IF ((P2Btn.P2M1_Tricolorlamp_Yellow AND NOT P2M1_DTSysState.bErrorStop AND NOT P2M1_WJSysState.bErrorStop AND NOT P2M1_WJSysState.bErrorStop AND
    P2Btn.P2M2_Tricolorlamp_Yellow AND NOT P2M2_DTSysState.bErrorStop AND NOT P2M2_WJSysState.bErrorStop AND NOT P2M2_WJSysState.bErrorStop AND
    P2Btn.P2M3_Tricolorlamp_Yellow AND NOT P2M3_DTSysState.bErrorStop AND NOT P2M3_WJSysState.bErrorStop AND NOT P2M3_WJSysState.bErrorStop ) OR 
	((P2M1_DTSysState.bErrorStop OR P2M1_WJSysState.bErrorStop OR P2M1_WJSysState.bErrorStop) AND
    (P2Btn.P2M2_Tricolorlamp_Yellow AND NOT P2M2_DTSysState.bErrorStop AND NOT P2M2_WJSysState.bErrorStop AND NOT P2M2_WJSysState.bErrorStop) AND
	(P2Btn.P2M3_Tricolorlamp_Yellow AND NOT P2M3_DTSysState.bErrorStop AND NOT P2M3_WJSysState.bErrorStop AND NOT P2M3_WJSysState.bErrorStop)) OR
	((P2Btn.P2M1_Tricolorlamp_Yellow AND NOT P2M1_DTSysState.bErrorStop AND NOT P2M1_WJSysState.bErrorStop AND NOT P2M1_WJSysState.bErrorStop) AND
	(P2M2_DTSysState.bErrorStop OR P2M2_WJSysState.bErrorStop OR P2M2_WJSysState.bErrorStop) AND	
	(P2Btn.P2M3_Tricolorlamp_Yellow AND NOT P2M3_DTSysState.bErrorStop AND NOT P2M3_WJSysState.bErrorStop AND NOT P2M3_WJSysState.bErrorStop)) OR
	((P2Btn.P2M1_Tricolorlamp_Yellow AND NOT P2M1_DTSysState.bErrorStop AND NOT P2M1_WJSysState.bErrorStop AND NOT P2M1_WJSysState.bErrorStop) AND
	(P2Btn.P2M2_Tricolorlamp_Yellow AND NOT P2M2_DTSysState.bErrorStop AND NOT P2M2_WJSysState.bErrorStop AND NOT P2M2_WJSysState.bErrorStop) AND
	(P2M3_DTSysState.bErrorStop OR P2M3_WJSysState.bErrorStop OR P2M3_WJSysState.bErrorStop) ) OR  Standby_TON.Q) AND
	NOT P2Btn.P2M1_Tricolorlamp_Green AND NOT P2Btn.P2M2_Tricolorlamp_Green AND NOT P2Btn.P2M3_Tricolorlamp_Green THEN
	 Status_switching2_TON.IN:=TRUE ;
	 Status_switching_TON.IN:=FALSE ;
END_IF

IF  Status_switching2_TON.Q THEN 
    P3Press.Device_Status_code:=18 ; //设备待机
END_IF	

Equipment_parameter_check_R(CLK:=Equipment_parameter_check=2  , Q=> ); //Equipment_parameter_check=1参数校验OK,Equipment_parameter_check=1参数校验NG
IF Equipment_parameter_check_R.Q THEN
   P3_Error[40]:=TRUE ;	//MES校验热压、称重、测厚参数报警，请检查参数设置s是否正确
   Equipment_parameter_check:=0 ;
END_IF

//xfp20240315 与MES交互优报表

ton2(IN:=NOT ton2.Q , PT:=T#5M , Q=> , ET=> );
IF ton2.Q THEN
   Mes1.uOther[0]:=1;
END_IF
ExcelRate_R(clk:=(Mes1.uOther[0]=1),Q=>);	//MES读取触发上升沿
MTDExcelRate_R(clk:=(MTD_Mes1.uOther[0]=2),Q=>);	//MTD完成上升沿
tonWaitMQdata(pt:=T#2S);
IF ExcelRate_R.Q THEN
	Mes1RdStep:=10;
END_IF	
CASE Mes1RdStep OF
	10:
		DTM_Mes1.uOther[0]:=1;
		Mes1RdStep:=20;
	20:	
		IF MTDExcelRate_R.Q THEN
			DTM_Mes1.uOther[0]:=0;
			Mes1RdStep:=30;
		END_IF
		IF NOT tonWaitMQdata.Q THEN
			tonWaitMQdata.IN:=TRUE;
		ELSE
			tonWaitMQdata.IN:=FALSE;
			Mes1.uOther[0]:=3;
			DTM_Mes1.uOther[0]:=0;
			Mes1RdStep:=0;	
		END_IF
	30:
		tonWaitMQdata.IN:=FALSE;
		IF system.stTime.wHour >=8 AND system.stTime.wHour <20 THEN
			Mes1.rExcelRate[0]:=1;	//班次，白班
			Mes1.rExcelRate[1]:=0;
			Mes1.rExcelRate[2]:=P3_Production.HMI_DayOkCount;	//生产良品数量
			Mes1.rExcelRate[3]:=P3_Production.HMI_DayNgCount;	//生产不良品数量
			Mes1.rExcelRate[4]:=P3_Production.HMI_DayQualified;	//良率			
			Mes1.rExcelRate[5]	:=MTD_Mes1.rExcelRate[0];
			Mes1.rExcelRate[6]	:=MTD_Mes1.rExcelRate[1];
			Mes1.rExcelRate[7]	:=MTD_Mes1.rExcelRate[2];
			Mes1.rExcelRate[8]	:=MTD_Mes1.rExcelRate[3];
			Mes1.rExcelRate[9]	:=MTD_Mes1.rExcelRate[4];
			Mes1.rExcelRate[10]	:=MTD_Mes1.rExcelRate[5];
			Mes1.rExcelRate[11]	:=MTD_Mes1.rExcelRate[6];
			Mes1.rExcelRate[12]	:=MTD_Mes1.rExcelRate[7];
			Mes1.rExcelRate[13]	:=MTD_Mes1.rExcelRate[8];
			Mes1.rExcelRate[14]	:=MTD_Mes1.rExcelRate[9];
			Mes1.rExcelRate[15]	:=MTD_Mes1.rExcelRate[10];
			Mes1.rExcelRate[16]	:=MTD_Mes1.rExcelRate[11];
			Mes1.rExcelRate[17]	:=MTD_Mes1.rExcelRate[12];
			Mes1.rExcelRate[18]	:=MTD_Mes1.rExcelRate[13];
			Mes1.rExcelRate[19]	:=MTD_Mes1.rExcelRate[14];
			Mes1.rExcelRate[20]	:=MTD_Mes1.rExcelRate[15];
			Mes1.rExcelRate[21]	:=MTD_Mes1.rExcelRate[16];
			Mes1.rExcelRate[22]	:=MTD_Mes1.rExcelRate[17];
			Mes1.rExcelRate[23]	:=MTD_Mes1.rExcelRate[18];
			Mes1.rExcelRate[24]	:=MTD_Mes1.rExcelRate[19];
			Mes1.rExcelRate[25]	:=MTD_Mes1.rExcelRate[20];
			Mes1.rExcelRate[26]	:=MTD_Mes1.rExcelRate[21];
			Mes1.rExcelRate[27]	:=MTD_Mes1.rExcelRate[22];
			Mes1.rExcelRate[28]	:=MTD_Mes1.rExcelRate[23];
			Mes1.rExcelRate[29]	:=MTD_Mes1.rExcelRate[24];
			Mes1.rExcelRate[30]	:=MTD_Mes1.rExcelRate[25];
			Mes1.rExcelRate[31]	:=MTD_Mes1.rExcelRate[26];			
			Mes1.rExcelRate[32]:=User01.P2M1_CCD.AnRec.DayNgclassification.X1_NG;	//叠台一正极X1纠偏轴不良数
			Mes1.rExcelRate[33]:=User01.P2M1_CCD.AnRec.DayNgclassification.X2_NG;	//叠台一正极X2纠偏轴不良数
			Mes1.rExcelRate[34]:=User01.P2M1_CCD.AnRec.DayNgclassification.Y_NG;	//叠台一正极Y纠偏轴不良数
			Mes1.rExcelRate[35]:=User01.P2M1_CCD.AnRec.DayNgclassification.R_NG;	//叠台一正极R角轮廓不良数
			Mes1.rExcelRate[36]:=User01.P2M1_CCD.AnRec.DayNgclassification.other_NG;	//叠台一正极其他类不良数
			Mes1.rExcelRate[37]:=User01.P2M2_CCD.AnRec.DayNgclassification.X1_NG;	//叠台二正极X1纠偏轴不良数
			Mes1.rExcelRate[38]:=User01.P2M2_CCD.AnRec.DayNgclassification.X2_NG;	//叠台二正极X2纠偏轴不良数
			Mes1.rExcelRate[39]:=User01.P2M2_CCD.AnRec.DayNgclassification.Y_NG;	//叠台二正极Y纠偏轴不良数
			Mes1.rExcelRate[40]:=User01.P2M2_CCD.AnRec.DayNgclassification.R_NG;	//叠台二正极R角轮廓不良数
			Mes1.rExcelRate[41]:=User01.P2M2_CCD.AnRec.DayNgclassification.other_NG;	//叠台二正极其他类不良数
			Mes1.rExcelRate[42]:=User01.P2M3_CCD.AnRec.DayNgclassification.X1_NG;	//叠台三正极X1纠偏轴不良数
			Mes1.rExcelRate[43]:=User01.P2M3_CCD.AnRec.DayNgclassification.X2_NG;	//叠台三正极X2纠偏轴不良数
			Mes1.rExcelRate[44]:=User01.P2M3_CCD.AnRec.DayNgclassification.Y_NG;	//叠台三正极Y纠偏轴不良数
			Mes1.rExcelRate[45]:=User01.P2M3_CCD.AnRec.DayNgclassification.R_NG;	//叠台三正极R角轮廓不良数
			Mes1.rExcelRate[46]:=User01.P2M3_CCD.AnRec.DayNgclassification.other_NG;	//叠台三正极其他类不良数
			//Mes1.rExcelRate[47]:=User01.P2M1_MachCtrl.DT_b.DT_DayHough_U;	//1#叠台OH不良，NG个数
			Mes1.rExcelRate[47]:=User01.P2M1_MachCtrl.DT_b.DT_DayHoughAn;		//1#叠台OH不良，正极NG数
			//Mes1.rExcelRate[49]:=User01.P2M2_MachCtrl.DT_b.DT_DayHough_U;	//2#叠台OH不良，NG个数
			Mes1.rExcelRate[49]:=User01.P2M2_MachCtrl.DT_b.DT_DayHoughAn;		//2#叠台OH不良，正极NG数
		//	Mes1.rExcelRate[51]:=User01.P2M3_MachCtrl.DT_b.DT_DayHough_U;	//3#叠台OH不良，NG个数
			Mes1.rExcelRate[51]:=User01.P2M3_MachCtrl.DT_b.DT_DayHoughAn;		//3#叠台OH不良，正极NG数
			Mes1.rExcelRate[53]:=P3_Production.NgPerHourDayCount[2];	//hi-potNG
			Mes1.rExcelRate[54]:=P3_Production.NgPerHourDayCount[4];	//厚度NG
			Mes1.rExcelRate[55]:=P3_Production.NgPerHourDayCount[6];	//烘烤超时NG
			Mes1.rExcelRate[56]:=P3_Production.NgPerHourDayCount[5];	//MESNG
			Mes1.rExcelRate[57]:=P3_Production.NgPerHourDayCount[1];	//扫码NG
			Mes1.rExcelRate[58]:=P3_Production.NgPerHourDayCount[3];	//其他不良	
			Mes1.rExcelRate[59]	:=MTD_Mes1.rExcelRate[27];
			Mes1.rExcelRate[60]	:=MTD_Mes1.rExcelRate[28];
			Mes1.rExcelRate[61]	:=MTD_Mes1.rExcelRate[29];
			Mes1.rExcelRate[62]	:=MTD_Mes1.rExcelRate[30];
			Mes1.rExcelRate[63]	:=MTD_Mes1.rExcelRate[31];
			Mes1.rExcelRate[64]	:=MTD_Mes1.rExcelRate[32];
			Mes1.rExcelRate[65]	:=MTD_Mes1.rExcelRate[33];
			Mes1.rExcelRate[66]	:=MTD_Mes1.rExcelRate[34];
			Mes1.rExcelRate[67]	:=MTD_Mes1.rExcelRate[35];
			Mes1.rExcelRate[68]	:=MTD_Mes1.rExcelRate[36];
			Mes1.rExcelRate[69]	:=MTD_Mes1.rExcelRate[37];
			Mes1.rExcelRate[70]	:=MTD_Mes1.rExcelRate[38];
			Mes1.rExcelRate[71]	:=MTD_Mes1.rExcelRate[39];
			Mes1.rExcelRate[72]	:=MTD_Mes1.rExcelRate[40];
			Mes1.rExcelRate[73]	:=MTD_Mes1.rExcelRate[41];
			Mes1.rExcelRate[74]	:=MTD_Mes1.rExcelRate[42];
			Mes1.rExcelRate[75]	:=MTD_Mes1.rExcelRate[43];
			Mes1.rExcelRate[76]	:=MTD_Mes1.rExcelRate[44];
			Mes1.rExcelRate[77]	:=MTD_Mes1.rExcelRate[45];
			Mes1.rExcelRate[78]	:=MTD_Mes1.rExcelRate[46];
			Mes1.rExcelRate[79]	:=MTD_Mes1.rExcelRate[47];
			Mes1.rExcelRate[80]	:=MTD_Mes1.rExcelRate[48];
			Mes1.rExcelRate[81]	:=MTD_Mes1.rExcelRate[49];
			Mes1.rExcelRate[82]	:=MTD_Mes1.rExcelRate[50];
			Mes1.rExcelRate[83]	:=MTD_Mes1.rExcelRate[51];
			Mes1.rExcelRate[84]	:=MTD_Mes1.rExcelRate[52];			
			Mes1.rExcelRate[85]:=User01.P2M1_CCD.CaRec.DayNgclassification.X1_NG;	//叠台一负极X1纠偏轴不良数
			Mes1.rExcelRate[86]:=User01.P2M1_CCD.CaRec.DayNgclassification.X2_NG;	//叠台一负极X2纠偏轴不良数
			Mes1.rExcelRate[87]:=User01.P2M1_CCD.CaRec.DayNgclassification.Y_NG;	//叠台一负极Y纠偏轴不良数
			Mes1.rExcelRate[88]:=User01.P2M1_CCD.CaRec.DayNgclassification.R_NG;	//叠台一负极R角轮廓不良数
			Mes1.rExcelRate[89]:=User01.P2M1_CCD.CaRec.DayNgclassification.other_NG;	//叠台一负极其他类不良数
			Mes1.rExcelRate[90]:=User01.P2M2_CCD.CaRec.DayNgclassification.X1_NG;	//叠台二负极X1纠偏轴不良数
			Mes1.rExcelRate[91]:=User01.P2M2_CCD.CaRec.DayNgclassification.X2_NG;	//叠台二负极X2纠偏轴不良数
			Mes1.rExcelRate[92]:=User01.P2M2_CCD.CaRec.DayNgclassification.Y_NG;	//叠台二负极Y纠偏轴不良数
			Mes1.rExcelRate[93]:=User01.P2M2_CCD.CaRec.DayNgclassification.R_NG;	//叠台二负极R角轮廓不良数
			Mes1.rExcelRate[94]:=User01.P2M2_CCD.CaRec.DayNgclassification.other_NG;	//叠台二负极其他类不良数
			Mes1.rExcelRate[95]:=User01.P2M3_CCD.CaRec.DayNgclassification.X1_NG;	//叠台三负极X1纠偏轴不良数
			Mes1.rExcelRate[96]:=User01.P2M3_CCD.CaRec.DayNgclassification.X2_NG;	//叠台三负极X2纠偏轴不良数
			Mes1.rExcelRate[97]:=User01.P2M3_CCD.CaRec.DayNgclassification.Y_NG;	//叠台三负极Y纠偏轴不良数
			Mes1.rExcelRate[98]:=User01.P2M3_CCD.CaRec.DayNgclassification.R_NG;	//叠台三负极R角轮廓不良数
			Mes1.rExcelRate[99]:=User01.P2M3_CCD.CaRec.DayNgclassification.other_NG;	//叠台三负极其他类不良数			
			Mes1.rExcelRate[100]:=User01.P2M1_MachCtrl.DT_b.DT_DayHoughCa;	//1#叠台OH不良负极NG数
			Mes1.rExcelRate[101]:=User01.P2M2_MachCtrl.DT_b.DT_DayHoughCa;	//2#叠台OH不良负极NG数
			Mes1.rExcelRate[102]:=User01.P2M3_MachCtrl.DT_b.DT_DayHoughCa;	//3#叠台OH不良负极NG数
			Mes1.rExcelRate[103]	:=MTD_Mes1.rExcelRate[53];			
			Mes1.rExcelRate[104]	:=MTD_Mes1.rExcelRate[54];	
			Mes1.rExcelRate[105]	:=MTD_Mes1.rExcelRate[55];			
			Mes1.rExcelRate[106]	:=MTD_Mes1.rExcelRate[56];	
			Mes1.rExcelRate[107]	:=MTD_Mes1.rExcelRate[57];			
			Mes1.rExcelRate[108]	:=MTD_Mes1.rExcelRate[58];	
			Mes1.rExcelRate[109]	:=(MTD_Mes1.rExcelRate[0]+MTD_Mes1.rExcelRate[15])/P2M1_Par.stDT_date.An_Quantity;		
			Mes1.rExcelRate[110]	:=(MTD_Mes1.rExcelRate[27]+MTD_Mes1.rExcelRate[41])/P2M1_Par.stDT_date.Ca_Quantity;			
			Mes1.uOther[0]:=2;	//plc数据写入完成
			Mes1RdStep:=0;
		ELSIF system.stTime.wHour >=20 OR system.stTime.wHour<8 THEN
			Mes1.rExcelRate[0]:=2;	//班次，夜班
			Mes1.rExcelRate[1]:=0;
			Mes1.rExcelRate[2]:=P3_Production.HMI_NightOkCount;	//生产良品数量
			Mes1.rExcelRate[3]:=P3_Production.HMI_NightNgCount;	//生产不良品数量
			Mes1.rExcelRate[4]:=P3_Production.HMI_NightQualified;	//良率			
			Mes1.rExcelRate[5]	:=MTD_Mes1.rExcelRate[0];
			Mes1.rExcelRate[6]	:=MTD_Mes1.rExcelRate[1];
			Mes1.rExcelRate[7]	:=MTD_Mes1.rExcelRate[2];
			Mes1.rExcelRate[8]	:=MTD_Mes1.rExcelRate[3];
			Mes1.rExcelRate[9]	:=MTD_Mes1.rExcelRate[4];
			Mes1.rExcelRate[10]	:=MTD_Mes1.rExcelRate[5];
			Mes1.rExcelRate[11]	:=MTD_Mes1.rExcelRate[6];
			Mes1.rExcelRate[12]	:=MTD_Mes1.rExcelRate[7];
			Mes1.rExcelRate[13]	:=MTD_Mes1.rExcelRate[8];
			Mes1.rExcelRate[14]	:=MTD_Mes1.rExcelRate[9];
			Mes1.rExcelRate[15]	:=MTD_Mes1.rExcelRate[10];
			Mes1.rExcelRate[16]	:=MTD_Mes1.rExcelRate[11];
			Mes1.rExcelRate[17]	:=MTD_Mes1.rExcelRate[12];
			Mes1.rExcelRate[18]	:=MTD_Mes1.rExcelRate[13];
			Mes1.rExcelRate[19]	:=MTD_Mes1.rExcelRate[14];
			Mes1.rExcelRate[20]	:=MTD_Mes1.rExcelRate[15];
			Mes1.rExcelRate[21]	:=MTD_Mes1.rExcelRate[16];
			Mes1.rExcelRate[22]	:=MTD_Mes1.rExcelRate[17];
			Mes1.rExcelRate[23]	:=MTD_Mes1.rExcelRate[18];
			Mes1.rExcelRate[24]	:=MTD_Mes1.rExcelRate[19];
			Mes1.rExcelRate[25]	:=MTD_Mes1.rExcelRate[20];
			Mes1.rExcelRate[26]	:=MTD_Mes1.rExcelRate[21];
			Mes1.rExcelRate[27]	:=MTD_Mes1.rExcelRate[22];
			Mes1.rExcelRate[28]	:=MTD_Mes1.rExcelRate[23];
			Mes1.rExcelRate[29]	:=MTD_Mes1.rExcelRate[24];
			Mes1.rExcelRate[30]	:=MTD_Mes1.rExcelRate[25];
			Mes1.rExcelRate[31]	:=MTD_Mes1.rExcelRate[26];			
			Mes1.rExcelRate[32]:=User01.P2M1_CCD.AnRec.NightNgclassification.X1_NG;	//叠台一正极X1纠偏轴不良数
			Mes1.rExcelRate[33]:=User01.P2M1_CCD.AnRec.NightNgclassification.X2_NG;	//叠台一正极X2纠偏轴不良数
			Mes1.rExcelRate[34]:=User01.P2M1_CCD.AnRec.NightNgclassification.Y_NG;	//叠台一正极Y纠偏轴不良数
			Mes1.rExcelRate[35]:=User01.P2M1_CCD.AnRec.NightNgclassification.R_NG;	//叠台一正极R角轮廓不良数
			Mes1.rExcelRate[36]:=User01.P2M1_CCD.AnRec.NightNgclassification.other_NG;	//叠台一正极其他类不良数
			Mes1.rExcelRate[37]:=User01.P2M2_CCD.AnRec.NightNgclassification.X1_NG;	//叠台二正极X1纠偏轴不良数
			Mes1.rExcelRate[38]:=User01.P2M2_CCD.AnRec.NightNgclassification.X2_NG;	//叠台二正极X2纠偏轴不良数
			Mes1.rExcelRate[39]:=User01.P2M2_CCD.AnRec.NightNgclassification.Y_NG;	//叠台二正极Y纠偏轴不良数
			Mes1.rExcelRate[40]:=User01.P2M2_CCD.AnRec.NightNgclassification.R_NG;	//叠台二正极R角轮廓不良数
			Mes1.rExcelRate[41]:=User01.P2M2_CCD.AnRec.NightNgclassification.other_NG;	//叠台二正极其他类不良数
			Mes1.rExcelRate[42]:=User01.P2M3_CCD.AnRec.NightNgclassification.X1_NG;	//叠台三正极X1纠偏轴不良数
			Mes1.rExcelRate[43]:=User01.P2M3_CCD.AnRec.NightNgclassification.X2_NG;	//叠台三正极X2纠偏轴不良数
			Mes1.rExcelRate[44]:=User01.P2M3_CCD.AnRec.NightNgclassification.Y_NG;	//叠台三正极Y纠偏轴不良数
			Mes1.rExcelRate[45]:=User01.P2M3_CCD.AnRec.NightNgclassification.R_NG;	//叠台三正极R角轮廓不良数
			Mes1.rExcelRate[46]:=User01.P2M3_CCD.AnRec.NightNgclassification.other_NG;	//叠台三正极其他类不良数
		//	Mes1.rExcelRate[47]:=User01.P2M1_MachCtrl.DT_b.DT_NightHough_U;	//1#叠台OH不良，NG个数
			Mes1.rExcelRate[47]:=User01.P2M1_MachCtrl.DT_b.DT_NightHoughAn;		//1#叠台OH不良，正极NG数
		//	Mes1.rExcelRate[49]:=User01.P2M2_MachCtrl.DT_b.DT_NightHough_U;	//2#叠台OH不良，NG个数
			Mes1.rExcelRate[49]:=User01.P2M2_MachCtrl.DT_b.DT_NightHoughAn;		//2#叠台OH不良，正极NG数
		//	Mes1.rExcelRate[51]:=User01.P2M3_MachCtrl.DT_b.DT_NightHough_U;	//3#叠台OH不良，NG个数
			Mes1.rExcelRate[51]:=User01.P2M3_MachCtrl.DT_b.DT_NightHoughAn;		//3#叠台OH不良，正极NG数
			Mes1.rExcelRate[53]:=P3_Production.NgPerHourNightCount[2];	//hi-potNG
			Mes1.rExcelRate[54]:=P3_Production.NgPerHourNightCount[4];	//厚度NG
			Mes1.rExcelRate[55]:=P3_Production.NgPerHourNightCount[6];	//烘烤超时NG
			Mes1.rExcelRate[56]:=P3_Production.NgPerHourNightCount[5];	//MESNG
			Mes1.rExcelRate[57]:=P3_Production.NgPerHourNightCount[1];	//扫码NG
			Mes1.rExcelRate[58]:=P3_Production.NgPerHourNightCount[3];	//其他不良	
			Mes1.rExcelRate[59]	:=MTD_Mes1.rExcelRate[27];
			Mes1.rExcelRate[60]	:=MTD_Mes1.rExcelRate[28];
			Mes1.rExcelRate[61]	:=MTD_Mes1.rExcelRate[29];
			Mes1.rExcelRate[62]	:=MTD_Mes1.rExcelRate[30];
			Mes1.rExcelRate[63]	:=MTD_Mes1.rExcelRate[31];
			Mes1.rExcelRate[64]	:=MTD_Mes1.rExcelRate[32];
			Mes1.rExcelRate[65]	:=MTD_Mes1.rExcelRate[33];
			Mes1.rExcelRate[66]	:=MTD_Mes1.rExcelRate[34];
			Mes1.rExcelRate[67]	:=MTD_Mes1.rExcelRate[35];
			Mes1.rExcelRate[68]	:=MTD_Mes1.rExcelRate[36];
			Mes1.rExcelRate[69]	:=MTD_Mes1.rExcelRate[37];
			Mes1.rExcelRate[70]	:=MTD_Mes1.rExcelRate[38];
			Mes1.rExcelRate[71]	:=MTD_Mes1.rExcelRate[39];
			Mes1.rExcelRate[72]	:=MTD_Mes1.rExcelRate[40];
			Mes1.rExcelRate[73]	:=MTD_Mes1.rExcelRate[41];
			Mes1.rExcelRate[74]	:=MTD_Mes1.rExcelRate[42];
			Mes1.rExcelRate[75]	:=MTD_Mes1.rExcelRate[43];
			Mes1.rExcelRate[76]	:=MTD_Mes1.rExcelRate[44];
			Mes1.rExcelRate[77]	:=MTD_Mes1.rExcelRate[45];
			Mes1.rExcelRate[78]	:=MTD_Mes1.rExcelRate[46];
			Mes1.rExcelRate[79]	:=MTD_Mes1.rExcelRate[47];
			Mes1.rExcelRate[80]	:=MTD_Mes1.rExcelRate[48];
			Mes1.rExcelRate[81]	:=MTD_Mes1.rExcelRate[49];
			Mes1.rExcelRate[82]	:=MTD_Mes1.rExcelRate[50];
			Mes1.rExcelRate[83]	:=MTD_Mes1.rExcelRate[51];
			Mes1.rExcelRate[84]	:=MTD_Mes1.rExcelRate[52];			
			Mes1.rExcelRate[85]:=User01.P2M1_CCD.CaRec.NightNgclassification.X1_NG;	//叠台一负极X1纠偏轴不良数
			Mes1.rExcelRate[86]:=User01.P2M1_CCD.CaRec.NightNgclassification.X2_NG;	//叠台一负极X2纠偏轴不良数
			Mes1.rExcelRate[87]:=User01.P2M1_CCD.CaRec.NightNgclassification.Y_NG;	//叠台一负极Y纠偏轴不良数
			Mes1.rExcelRate[88]:=User01.P2M1_CCD.CaRec.NightNgclassification.R_NG;	//叠台一负极R角轮廓不良数
			Mes1.rExcelRate[89]:=User01.P2M1_CCD.CaRec.NightNgclassification.other_NG;	//叠台一负极其他类不良数
			Mes1.rExcelRate[90]:=User01.P2M2_CCD.CaRec.NightNgclassification.X1_NG;	//叠台二负极X1纠偏轴不良数
			Mes1.rExcelRate[91]:=User01.P2M2_CCD.CaRec.NightNgclassification.X2_NG;	//叠台二负极X2纠偏轴不良数
			Mes1.rExcelRate[92]:=User01.P2M2_CCD.CaRec.NightNgclassification.Y_NG;	//叠台二负极Y纠偏轴不良数
			Mes1.rExcelRate[93]:=User01.P2M2_CCD.CaRec.NightNgclassification.R_NG;	//叠台二负极R角轮廓不良数
			Mes1.rExcelRate[94]:=User01.P2M2_CCD.CaRec.NightNgclassification.other_NG;	//叠台二负极其他类不良数
			Mes1.rExcelRate[95]:=User01.P2M3_CCD.CaRec.NightNgclassification.X1_NG;	//叠台三负极X1纠偏轴不良数
			Mes1.rExcelRate[96]:=User01.P2M3_CCD.CaRec.NightNgclassification.X2_NG;	//叠台三负极X2纠偏轴不良数
			Mes1.rExcelRate[97]:=User01.P2M3_CCD.CaRec.NightNgclassification.Y_NG;	//叠台三负极Y纠偏轴不良数
			Mes1.rExcelRate[98]:=User01.P2M3_CCD.CaRec.NightNgclassification.R_NG;	//叠台三负极R角轮廓不良数
			Mes1.rExcelRate[99]:=User01.P2M3_CCD.CaRec.NightNgclassification.other_NG;	//叠台三负极其他类不良数			
			Mes1.rExcelRate[100]:=User01.P2M1_MachCtrl.DT_b.DT_NightHoughCa;	//1#叠台OH不良负极NG数
			Mes1.rExcelRate[101]:=User01.P2M2_MachCtrl.DT_b.DT_NightHoughCa;	//2#叠台OH不良负极NG数
			Mes1.rExcelRate[102]:=User01.P2M3_MachCtrl.DT_b.DT_NightHoughCa;	//3#叠台OH不良负极NG数
			Mes1.rExcelRate[103]	:=MTD_Mes1.rExcelRate[53];			
			Mes1.rExcelRate[104]	:=MTD_Mes1.rExcelRate[54];	
			Mes1.rExcelRate[105]	:=MTD_Mes1.rExcelRate[55];			
			Mes1.rExcelRate[106]	:=MTD_Mes1.rExcelRate[56];	
			Mes1.rExcelRate[107]	:=MTD_Mes1.rExcelRate[57];			
			Mes1.rExcelRate[108]	:=MTD_Mes1.rExcelRate[58];		
     		Mes1.rExcelRate[109]	:=(MTD_Mes1.rExcelRate[0]+MTD_Mes1.rExcelRate[15])/P2M1_Par.stDT_date.An_Quantity;		
			Mes1.rExcelRate[110]	:=(MTD_Mes1.rExcelRate[27]+MTD_Mes1.rExcelRate[41])/P2M1_Par.stDT_date.Ca_Quantity;	;		
			Mes1.uOther[0]:=2;	//plc数据写入完成
			Mes1RdStep:=0;
		END_IF	
END_CASE


//功能开关状态
Mes1.bFuncEN[1]:=MTD_Mes1.bFuncEN[1];//模切段CCD通讯开关状态
Mes1.bFuncEN[2]:=MTD_Mes1.bFuncEN[2];//线扫CCD开关状态
Mes1.bFuncEN[3]:=MTD_Mes1.bFuncEN[3];//冲R角定位开关状态
Mes1.bFuncEN[4]:=MTD_Mes1.bFuncEN[4];//裁切定位开关状态
Mes1.bFuncEN[5]:=MTD_Mes1.bFuncEN[5];//尺寸检测开关状态
Mes1.bFuncEN[6]:=MTD_Mes1.bFuncEN[6];//物料校验功能开关状态
Mes1.bFuncEN[7]:=MTD_Mes1.bFuncEN[7];//来料不良检测开关状态
Mes1.bFuncEN[8]:=P2M1_Par.iModeEN.CCD_ChosesHMIEN;//一叠台CCD通讯开关状态
Mes1.bFuncEN[9]:=P2M2_Par.iModeEN.CCD_ChosesHMIEN;
Mes1.bFuncEN[10]:=P2M3_Par.iModeEN.CCD_ChosesHMIEN;
Mes1.bFuncEN[11]:=P2M1_Par.iModeEN.DT_CCD_TwoModelEN;//一叠台CCD复检开关状态
Mes1.bFuncEN[12]:=P2M2_Par.iModeEN.DT_CCD_TwoModelEN;
Mes1.bFuncEN[13]:=P2M3_Par.iModeEN.DT_CCD_TwoModelEN;
Mes1.bFuncEN[14]:=P2M1_Par.iModeEN.DT_OverhangEN;//一叠台对齐度开关状态
Mes1.bFuncEN[15]:=P2M2_Par.iModeEN.DT_OverhangEN;
Mes1.bFuncEN[16]:=P2M3_Par.iModeEN.DT_OverhangEN;
Mes1.bFuncEN[17]:=P2M1_Par.iModeEN.DT_CellNG_TFEN;//一叠台对齐度踢废开关状态
Mes1.bFuncEN[18]:=P2M2_Par.iModeEN.DT_CellNG_TFEN;
Mes1.bFuncEN[19]:=P2M3_Par.iModeEN.DT_CellNG_TFEN;
Mes1.bFuncEN[20]:=P2M1_MachCtrl.DT_b.PartNumberOff;//一叠台MES物料码校验开关状态
Mes1.bFuncEN[21]:=P2M2_MachCtrl.DT_b.PartNumberOff;
Mes1.bFuncEN[22]:=P2M3_MachCtrl.DT_b.PartNumberOff;
Mes1.bFuncEN[23]:=P2M1_MachCtrl.DT_b.Yellowmark_TF;//一叠台隔膜色标开关状态
Mes1.bFuncEN[24]:=P2M2_MachCtrl.DT_b.Yellowmark_TF;
Mes1.bFuncEN[25]:=P2M3_MachCtrl.DT_b.Yellowmark_TF;
Mes1.bFuncEN[26]:=P3User2_Par.Shield[1];//短路测试开关状态
Mes1.bFuncEN[27]:=P3User2_Par.Shield[2];//称重测试开关状态
Mes1.bFuncEN[28]:=P3User2_Par.Shield[3];//测厚测试开关状态
Mes1.bFuncEN[29]:=P3User2_Par.Shield[8];//后段条码校验开关状态

DTM_Mes1.bFuncEN[0]:=P3User2_Par.Shield[5];
DTM_Mes1.bFuncEN[1]:=Mes1.Error[1];
DTM_Mes1.bFuncEN[2]:=Mes1.Error[2];
DTM_Mes1.bFuncEN[3]:=Mes1.Error[3];
DTM_Mes1.bFuncEN[4]:=Mes1.Error[4];
DTM_Mes1.bFuncEN[5]:=Mes1.Error[5];
DTM_Mes1.bFuncEN[6]:=Mes1.Error[6];
DTM_Mes1.bFuncEN[7]:=Mes1.Error[7];

IF stSysState.hmiReset THEN
	MEMSET(ADR(Mes1.Error),0,SIZEOF(Mes1.Error)); 
END_IF

END_PROGRAM

// ---- P3POUs/POUs/Auxiliary/LateBlanking_Tips.TcPOU
PROGRAM LateBlanking_Tips
VAR
	
END_VAR

////////////////////////////提示不停机

//冷压上料提示
IF  Step30=35 AND (NOT arrAxisCtrl[P2AxisNo.P2M1_GluingLine].Cmd.arrbRealPoint[9] OR NOT arrAxisCtrl[P2AxisNo.P2M1_GluingWhirling].Cmd.arrbRealPoint[6]) AND arrAxisCtrl[P2AxisNo.P2M1_GluingLine].Status.NoMoving 
	AND arrAxisCtrl[P2AxisNo.P2M1_GluingLine].Status.Homed AND arrAxisCtrl[P2AxisNo.P2M1_GluingWhirling].Status.NoMoving  AND arrAxisCtrl[P2AxisNo.P2M1_GluingWhirling].Status.Homed THEN
		tip_1[1]:=TRUE;//一号叠台侧贴胶平移不在下电芯位或者侧贴胶旋转不在下电芯位
	ELSE
		tip_1[1]:=FALSE;	
END_IF
	
IF  Step30=1035 AND (NOT arrAxisCtrl[P2AxisNo.P2M1_GluingLine].Cmd.arrbRealPoint[9] OR NOT arrAxisCtrl[P2AxisNo.P2M1_GluingWhirling].Cmd.arrbRealPoint[6]) AND arrAxisCtrl[P2AxisNo.P2M1_GluingLine].Status.NoMoving 
	AND arrAxisCtrl[P2AxisNo.P2M1_GluingLine].Status.Homed AND arrAxisCtrl[P2AxisNo.P2M1_GluingWhirling].Status.NoMoving  AND arrAxisCtrl[P2AxisNo.P2M1_GluingWhirling].Status.Homed THEN
		tip_1[2]:=TRUE;//二号叠台侧贴胶平移不在下电芯位或者侧贴胶旋转不在下电芯位
	ELSE
		tip_1[2]:=FALSE;	
END_IF	

IF   Step30=2035 AND (NOT arrAxisCtrl[P2AxisNo.P2M3_GluingLine].Cmd.arrbRealPoint[9] OR NOT arrAxisCtrl[P2AxisNo.P2M3_GluingWhirling].Cmd.arrbRealPoint[6])
	 AND arrAxisCtrl[P2AxisNo.P2M3_GluingLine].Status.NoMoving AND arrAxisCtrl[P2AxisNo.P2M3_GluingLine].Status.Homed  AND arrAxisCtrl[P2AxisNo.P2M3_GluingWhirling].Status.NoMoving  
	 AND arrAxisCtrl[P2AxisNo.P2M3_GluingWhirling].Status.Homed  THEN
		tip_1[3]:=TRUE;//三号叠台侧贴胶平移不在下电芯位或者侧贴胶旋转不在下电芯位
	ELSE
		tip_1[3]:=FALSE;	
END_IF	

IF Step30=3035 AND PermitColdPressRack AND arrAxisCtrl[P3AxisNo.P3M1_ColdpreActuated].Cmd.arrbRealPoint[1] AND arrAxisCtrl[P3AxisNo.P3M1_ColdpreActuated].Status.NoMoving 
	AND NOT arrAxisCtrl[P3AxisNo.P3M1_ColdpreSupPlateLine].Cmd.arrbRealPoint[1] AND arrAxisCtrl[P3AxisNo.P3M1_ColdpreSupPlateLine].Status.NoMoving THEN
		tip_1[4]:=TRUE;//冷压上料时托板不在初始位
	ELSE
		tip_1[4]:=FALSE;	
END_IF	

IF SingleStep[1] THEN
		tip_1[5]:=TRUE;//冷压上料单步中
	ELSE
		tip_1[5]:=FALSE;
END_IF

IF (P2Senser.P2M1_Securitydoorswitch3 AND P2Senser.P2M1_Securitydoorswitch4
	AND P2Senser.P2M2_Securitydoorswitch3 AND P2Senser.P2M2_Securitydoorswitch4
	AND P2Senser.P2M3_Securitydoorswitch3 AND P2Senser.P2M3_Securitydoorswitch4) THEN
		tip_1[6]:=FALSE;//叠片冷压上料门禁
	ELSE
		tip_1[6]:=TRUE; 
END_IF

/////冷压提示
IF   Step31=30 AND (arrAxisCtrlV2[P3AxisNo.P3_M2_OvenRetracting].Cmd.arrbRealPoint[43] OR LREAL_TO_REAL(arrAxisCtrlV2[P3AxisNo.P3_M2_OvenCarrying].Status.fActPos)>arrAxisParV2[P3AxisNo.P3_M2_OvenCarrying].arrTargetPoint[44]) AND 
    (arrAxisCtrl[P3AxisNo.P3M1_ColdpreRetracting].Cmd.arrbRealPoint[1] OR LREAL_TO_REAL(arrAxisCtrl[P3AxisNo.P3M1_ColdpreLine].Status.fActPos)>=arrAxisPar[P3AxisNo.P3M1_ColdpreLine].arrTargetPoint[1]) AND 
	arrAxisCtrl[P3AxisNo.P3M1_ColdpreSupPlateLine].Cmd.arrbRealPoint[2] AND arrAxisCtrl[P3AxisNo.P3M1_ColdpreSupPlateLine].Status.NoMoving 
	 AND Permit_Cold_Press AND NOT b_Press_condition[1] AND CellMemory[CellNo.Coldpress].Cell THEN	
		tip_2[1]:=TRUE;//冷压未感应到电芯报警
	ELSE
		tip_2[1]:=FALSE;
END_IF

IF SingleStep[2] THEN
		tip_2[2]:=TRUE;//冷压单步中
	ELSE
		tip_2[2]:=FALSE;
END_IF

/////烤箱上下料提示
IF  (LREAL_TO_REAL(arrAxisCtrl[P3AxisNo.P3_M4_WeighLine].Status.fActPos)>WeighLine_1 OR NOT arrAxisCtrl[P3AxisNo.P3_M4_WeighWhirling].Cmd.arrbRealPoint[3])
	AND PermitHotPressRack AND arrAxisCtrl[P3AxisNo.P3_M4_WeighLine].Status.Homed AND Step32=53 AND arrAxisCtrl[P3AxisNo.P3_M4_WeighWhirling].Status.NoMoving THEN
		tip_3[1]:=TRUE;//烤箱准备下料时，称重平移不在初始位或者称重旋转不在称重位
	ELSE
		tip_3[1]:=FALSE;
END_IF

IF (LREAL_TO_REAL(arrAxisCtrl[P3AxisNo.P3_M4_WeighLine].Status.fActPos)>WeighLine_1 OR NOT arrAxisCtrl[P3AxisNo.P3_M4_WeighWhirling].Cmd.arrbRealPoint[3]) AND Step32=105 THEN
		tip_3[1]:=TRUE;//烤箱准备下料时，称重平移不在初始位或者称重旋转不在称重位
	ELSE
		tip_3[1]:=FALSE;
END_IF

IF (LREAL_TO_REAL(arrAxisCtrl[P3AxisNo.P3_M4_WeighLine].Status.fActPos)>WeighLine_1 OR NOT arrAxisCtrl[P3AxisNo.P3_M4_WeighWhirling].Cmd.arrbRealPoint[3]) AND Step32=1115 THEN
		tip_3[2]:=TRUE;//烤箱上料时，称重平移不在初始位或者称重旋转不在称重位
	ELSE
		tip_3[2]:=FALSE;
END_IF

IF SingleStep[3] THEN
		tip_3[3]:=TRUE;//烤箱上下料单步中
	ELSE
		tip_3[3]:=FALSE;
END_IF









/////热压提示
IF  Step33=30 AND (arrAxisCtrlV2[P3AxisNo.P3_M2_OvenRetracting].Cmd.arrbRealPoint[43] OR LREAL_TO_REAL(arrAxisCtrlV2[P3AxisNo.P3_M2_OvenCarrying].Status.fActPos)<arrAxisParV2[P3AxisNo.P3_M2_OvenCarrying].arrTargetPoint[45]) AND 
     arrAxisCtrl[P3AxisNo.P3_M4_WeighLine].Cmd.arrbRealPoint[1] AND arrAxisCtrl[P3AxisNo.P3_M3_HotPressingLine].Cmd.arrbRealPoint[2] AND arrAxisCtrl[P3AxisNo.P3_M3_HotPressingLine].Status.NoMoving 
	AND Permit_Hot_Press  AND NOT b_Press_condition[2] AND CellMemory[CellNo.Hotpress].Cell THEN
		tip_4[1]:=TRUE;//热压未感应到电芯报警
	ELSE
		tip_4[1]:=FALSE;
END_IF

IF SingleStep[4] THEN
		tip_4[2]:=TRUE;//热压单步中
	ELSE
		tip_4[2]:=FALSE;
END_IF


////称重上料提示
IF SingleStep[5] THEN
		tip_5[1]:=TRUE;//称重上料单步中
	ELSE
		tip_5[1]:=FALSE;
END_IF





//分选提示
IF SingleStep[6] THEN
		tip_6[1]:=TRUE;//分选单步中
	ELSE
		tip_6[1]:=FALSE;
END_IF





//下料提示
IF SingleStep[7] THEN
		tip_7[1]:=TRUE;//下料单步中
	ELSE
		tip_7[1]:=FALSE;
END_IF

END_PROGRAM

// ---- P3POUs/POUs/Auxiliary/MQ_FSY.TcPOU
PROGRAM MQ_FSY
VAR
//	CS_FSY_TcpAn: CS_FsyTcp;
	CS_FSY_TcpCa: CS_FsyTcp;
	Cold_step :UINT;
	scan_TON1 :Tc2_Standard.TON;
	Scan_TON :ARRAY[1..7] OF Tc2_Standard.TON;
	Scan_code_Z : R_TRIG;
	I:INT;
END_VAR

//扫码



Saoma();
P3User2_Par.MQ_AnFSY_IP:='192.168.10.40';
P3User2_Par.MQ_CaFSY_IP:='192.168.10.41';
Scan_TON[1](PT:=T#1MS);
Scan_TON[2](PT:=T#1MS);
Scan_TON[3](PT:=T#1MS);
Scan_TON[4](PT:=T#100MS);

Scan_code_Z (CLK:=Cold_Scan_code, Q=>);

IF Scan_code_Z.Q AND  Cold_step=0 THEN
	 Cold_step:=10;
END_IF




CASE Cold_step OF
0:
	IF Scan_start AND NOT bCodeError AND NOT bCodeConError AND NOT P3User2_Par.Shield[4] THEN
	 Cold_step:=10;
	 Code_State:=0;
	ELSIF P3User2_Par.Shield[4] THEN
	 Cold_step:=70;
	END_IF
10:
	Scan_TON[1].IN:=FALSE;
	Scan_TON[2].IN:=FALSE;
	Scan_TON[3].IN:=FALSE;
	Cold_step:=20;
	
20:
	bScan_init:=TRUE;
	Scan_TON[1].IN:=TRUE;
	IF Scan_TON[1].Q THEN
		bScan_init:=FALSE;
		Scan_TON[1].IN:=FALSE;
		Cold_step:=30;
	END_IF

30:
	bTcpOpen:=TRUE;
	Scan_TON[2].IN:=TRUE;
	IF Scan_TON[2].Q THEN
		bTcpOpen:=FALSE;
		Scan_TON[2].IN:=FALSE;
		Cold_step:=40;
	END_IF

40:
	IF bTcpOpen_OK THEN
		Cold_step:=50;
	END_IF

50:
	bScan_start:=TRUE;
	Scan_TON[3].IN:=TRUE;
	IF Scan_TON[3].Q THEN
		bScan_start:=FALSE;
		Scan_TON[3].IN:=FALSE;
		Cold_step:=60;
	END_IF
60:
	Scan_TON[4].IN:=TRUE;
	IF 	Scan_TON[4].Q THEN
		Cold_step:=70;
		Scan_TON[4].IN:=FALSE;
	END_IF

70:
IF NOT P3User2_Par.Shield[4] THEN
	IF Code_State=1 AND (strCode<>'') THEN
		CellMemory[CellNo.OvenMoveClip1].Cell_number1:=strCode;
		IF strCode=CellMemory[CellNo.OvenMoveClip1].Cell_number THEN
			CellMemory[CellNo.OvenMoveClip1].ScanCode:=1;
			Scan_start:=FALSE;
			Scan_finish:=TRUE;
			Cold_step:=80;				
			I:=0;
		ELSIF strCode<>CellMemory[CellNo.OvenMoveClip1].Cell_number THEN
			CellMemory[CellNo.OvenMoveClip1].ScanCode:=2;
			P3_Error[79]:=TRUE;//冷压扫码第二次扫码校验NG
			Scan_start:=FALSE;
			Scan_finish:=TRUE;
			Cold_step:=80;
			I:=0;
		END_IF
	ELSIF  Code_State=2 AND I<3 THEN
			Cold_step:=10;
			I:=I+1;		
	ELSIF Code_State=2 AND I>=3 THEN
		CellMemory[CellNo.ColdpressClip].Cell_number1:=strCode;
		CellMemory[CellNo.ColdpressClip].ScanCode:=2;
		P3_Error[16]:=TRUE;//冷压扫码NG报警
		Scan_start:=FALSE;
		Scan_finish:=TRUE;
		Cold_step:=80;
		I:=0;
	END_IF
ELSIF P3User2_Par.Shield[4] THEN
		CellMemory[CellNo.OvenMoveClip1].Cell_number1:='A1234567890ABCDEF';
		CellMemory[CellNo.OvenMoveClip1].ScanCode:=1;
		Scan_start:=FALSE;
		Scan_finish:=TRUE;
		Cold_step:=80;				
		I:=0;
END_IF
80:
	IF NOT Scan_finish THEN
		Cold_step:=0;
	END_IF
END_CASE

ACTION Saoma:
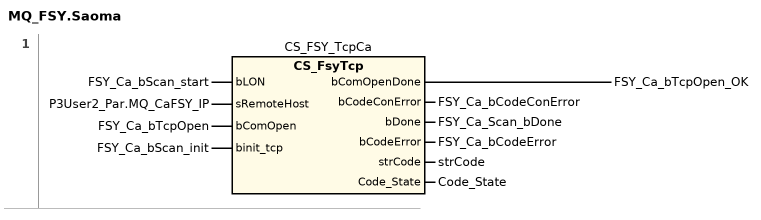
// NETWORK 1
CS_FSY_TcpCa(
    bLON := FSY_Ca_bScan_start,
    sRemoteHost := P3User2_Par.MQ_CaFSY_IP,
    bComOpen := FSY_Ca_bTcpOpen,
    binit_tcp := FSY_Ca_bScan_init,
    bCodeConError => FSY_Ca_bCodeConError,
    bDone => FSY_Ca_Scan_bDone,
    bCodeError => FSY_Ca_bCodeError,
    strCode => strCode,
    Code_State => Code_State); // CS_FsyTcp
FSY_Ca_bTcpOpen_OK := CS_FSY_TcpCa.bComOpenDone;
END_ACTION

END_PROGRAM

// ---- P2POUs/BasicFunction/10_MES/CS_FsyTcp.TcPOU
FUNCTION_BLOCK PUBLIC CS_FsyTcp
VAR_INPUT
	bLON                           :BOOL; 	//  扫码开
	sRemoteHost: T_IPv4Addr; 			//扫码枪IP地址;
	bComOpen                  :BOOL; 	 //扫码Tcp 开
	binit_tcp:BOOL;							//功能块初始化，所有状态全部清零；
END_VAR

VAR_OUTPUT
	bComOpenDone          :BOOL;  //扫码Tcp 打开OK
    bCodeConError             :BOOL;//扫码通讯故障
	bDone                         :BOOL; //扫码完成
    bCodeError                  :BOOL;//扫码故障	
    strCode                       :STRING;//条码结果
	Code_State						:INT;//扫码结果 1：OK  2：NG
END_VAR

VAR_IN_OUT

END_VAR

VAR
	bLOFF                          :BOOL; 	//扫码关	
	bComClose                  :BOOL;  	//扫码Tcp 关
	fbTcpCon:FB_SocketConnect;
	fbTcpSend:FB_SocketSend;
	fbTcpRec:FB_SocketReceive;
	fbTcpClose: FB_SocketClose;
	bConnect: BOOL;//打开TCP连接;
	bClose: BOOL;		//关闭TCP连接;
	hTcpSock: T_HSOCKET;
	StrSend: STRING;
	StrReceive: ARRAY[0..255]OF BYTE; 
	StrReceive2:STRING:='';//clean;
	fbUdpCreate:FB_SocketUdpCreate;
	hUdp: T_HSOCKET;
	bCreate: BOOL;
	port: UDINT:=23;
	bSendTcp: BOOL;
	bReceiveTcp: BOOL;
	bAcceptTcp: BOOL;
	fbSwingHalt2: MC_Halt;
    TON01:TON;
	Lenth: UINT;
	StrSend2: STRING;
	bSendTcp2: BOOL;
	iComSetp: INT;
	bRectiveEN: BOOL;
	TON_3: Ton;
	TON_4: TON;
	tTon5: BOOL;
	TON_5: TON;
	TON_6: TON;
	TCP_IP_Lis: FB_SocketListen;
	TCP_IP_SocketAccept: FB_SocketAccept;
	Listener: T_HSOCKET;
	blisten: BOOL;
	closeall_do: BOOL;
	LocalPort: UDINT;
	 closeall:FB_SocketCloseAll;
END_VAR




	Config();
	
	M_SendReceive();

ACTION Config:
TON_3(IN:=binit_tcp , PT:=T#2MS , Q=> , ET=> ); 
IF binit_tcp THEN
	iComSetp:=0;
	bComOpenDone:=FALSE;
    bCodeConError:=FALSE;
	bCodeError:=FALSE;
	bConnect:=FALSE;
	bClose :=TRUE;
	bDone:=FALSE;
    strCode:=StrReceive2;	 
//	StrReceive:=StrReceive2;	 
	Code_State:=0;
	bRectiveEN:=FALSE;
	bSendTcp:=FALSE;
END_IF
IF TON_3.Q THEN
	binit_tcp:=FALSE;
	bClose :=FALSE;
END_IF
fbTcpClose(
	sSrvNetId:= ''   , 
	hSocket:=hTcpSock , 
	bExecute:=bClose , 
	tTimeout:=T#2S , 
	bBusy=> , 
	bError=> , 
	nErrId=> );	
fbTcpClose(
	sSrvNetId:= ''   , 
	hSocket:=Listener , 
	bExecute:=bClose , 
	tTimeout:=T#2S , 
	bBusy=> , 
	bError=> , 
	nErrId=> );	
TCP_IP_Lis(
	sSrvNetId:= , 
	sLocalHost:='192.168.10.10', 
	nLocalPort:=LocalPort, 
	bExecute:=bConnect, 
	tTimeout:=T#2S , 
	bBusy=> , 
	bError=> , 
	nErrId=> , 
	hListener=>Listener );
///////////////////////////////////
Listener.handle;
Listener.localAddr;
Listener.remoteAddr; 
///////////////////////////////////
TCP_IP_SocketAccept(
	sSrvNetId:= , 
	hListener:=Listener , 
	bExecute:=bAcceptTcp , 
	tTimeout:=T#2S , 
	bAccepted=> , 
	bBusy=> , 
	bError=> , 
	nErrId=> , 
	hSocket=>hTcpSock );	

hTcpSock.handle;
hTcpSock.localAddr;
hTcpSock.remoteAddr;
IF bComOpen THEN
    bComOpenDone:=FALSE;
    bCodeConError:=FALSE;
    iComSetp:=100;
END_IF
 IF bComClose THEN
    bComOpenDone:=FALSE;
    bCodeConError:=FALSE;
     iComSetp:=200;
END_IF 

 CASE iComSetp OF 
   100:
	   bConnect:=TRUE;	
	   bClose:=FALSE;
	   bComOpen:=FALSE;
	   iComSetp:=110;
  110:
	  IF bConnect  THEN
		  bConnect:=FALSE;	
		   iComSetp:=120;
	  ELSIF fbTcpCon.bError THEN
		  iComSetp:=999;
	 END_IF
  120:
	 IF TCP_IP_Lis.hListener.handle>0  THEN
		bComOpenDone:=TRUE;//扫码枪连接成功；
		 iComSetp:=666;
	 ELSIF  NOT fbTcpCon.bBusy AND fbTcpCon.hSocket.handle=0  THEN
		iComSetp:=999;
	 END_IF

  200:
	   bConnect:=FALSE;	
	   bClose:=TRUE;
	   bComClose:=FALSE;
       iComSetp:=210;
  210:
	  IF fbTcpClose.bBusy THEN
		  bConnect:=FALSE;	
		   iComSetp:=666;
	 END_IF
  
  999:
	   bCodeConError:=TRUE;
	   iComSetp:=0;
END_CASE




 //发送； 
fbTcpSend(
		sSrvNetId:= , 
		hSocket:=hTcpSock , 
		cbLen:=SIZEOF(StrSend), 
		pSrc:= ADR(StrSend), 
		bExecute:= bSendTcp, 
		tTimeout:= T#5S , 
		bBusy=> , 
		bError=> , 
		nErrId=> );

//接收
	TON_6(IN:=NOT TON_6.Q AND fbTcpCon.hSocket.handle>0, PT:=T#3S , Q=> , ET=> );
	IF TON_6.Q THEN
		bReceiveTcp := NOT bReceiveTcp;
	END_IF
fbTcpRec(
	sSrvNetId:= , 
	hSocket:= hTcpSock, 
	cbLen:=SIZEOF(StrReceive) , 
	pDest:=ADR(StrReceive) , 
	bExecute:=bReceiveTcp , 
	tTimeout:= T#5S, 
	bBusy=> , 
	bError=> , 
	nErrId=> , 
	nRecBytes=> );	
	
CloseAll(
	sSrvNetId:= ,
	bExecute:=closeall_do ,
	tTimeout:= , 
	bBusy=> , 
	bError=> , 
	nErrId=> );
END_ACTION

ACTION M_SendReceive:

END_ACTION

END_FUNCTION_BLOCK

// ---- P2POUs/BasicFunction/08_Data/FB_DTData.TcPOU
FUNCTION_BLOCK FB_DTData
VAR_INPUT
    Alm :    BOOL ;//报警
	Wait :BOOL ;//待机
	Run :BOOL ;//运行
	Overhang_NG:BOOL ;//对齐度NG下料
	GM_change:BOOL ;//隔膜更换时间
	Query:BOOL;//时间查询
	
END_VAR

VAR_OUTPUT
	STTimedata:ARRAY[0..32] OF ST_Timedata;
END_VAR

VAR
	
	rRun : R_TRIG;
	rAlm : R_TRIG;
	rWait : R_TRIG;
	rOverhang_NG : R_TRIG;
	rGM_change: R_TRIG;
	fRun: F_TRIG;
	fAlm: F_TRIG;
	fWait: F_TRIG;
	fOverhang_NG: F_TRIG;
	fGM_change: F_TRIG;
	delay:BOOL ;//延时
	TON_1: TON;
	i:INT;
	K: INT;
	J: BOOL;
END_VAR

VAR_IN_OUT
     date1:INT;//查询日期
END_VAR



K:=K+1;
	IF K>499THEN
		J:=TRUE;
		K:=0;
	ELSE
		J:=FALSE;
	END_IF


///////////////运行时间/////////////////
//rRun(CLK:= Pulse._500ms.Q , Q=> );
rRun(CLK:= J , Q=> );

IF rRun.Q  AND  Run THEN
	STTimedata[system.stTime.wDay].RunTime[system.stTime.wHour]:=STTimedata[system.stTime.wDay].RunTime[system.stTime.wHour]+1;
END_IF

IF STTimedata[system.stTime.wDay].RunTime[system.stTime.wHour]> 3600 THEN
	STTimedata[system.stTime.wDay].RunTime[system.stTime.wHour]:= 3600 ;
END_IF

//IF STTimedata[system.stTime.wDay].AlmTime[system.stTime.wHour]= 0 AND STTimedata[system.stTime.wDay].WaitTime[system.stTime.wHour]= 0  AND 
  //  (STTimedata[system.stTime.wDay].RunTime[system.stTime.wHour]= 3585  OR  STTimedata[system.stTime.wDay].RunTime[system.stTime.wHour]= 3586 ) THEN
	//STTimedata[system.stTime.wDay].RunTime[system.stTime.wHour]:= 3600 ;
//END_IF

///////////////待机时间///////////////
rWait(CLK:=J , Q=> );

IF rWait.Q  AND Wait THEN
	STTimedata[system.stTime.wDay].WaitTime[system.stTime.wHour]:=STTimedata[system.stTime.wDay].WaitTime[system.stTime.wHour]+1;
END_IF
 
IF STTimedata[system.stTime.wDay].WaitTime[system.stTime.wHour]> 3600 THEN
	STTimedata[system.stTime.wDay].WaitTime[system.stTime.wHour]:= 3600 ;
END_IF

//IF STTimedata[system.stTime.wDay].RunTime[system.stTime.wHour]= 0 AND STTimedata[system.stTime.wDay].AlmTime[system.stTime.wHour]= 0  AND
  //  (STTimedata[system.stTime.wDay].RunTime[system.stTime.wHour]= 3585  OR  STTimedata[system.stTime.wDay].RunTime[system.stTime.wHour]= 3586 )  THEN
//	STTimedata[system.stTime.wDay].WaitTime[system.stTime.wHour]:= 3600 ;
//END_IF

////////////////报警时间///////////////
rAlm(CLK:=J , Q=> );

IF rAlm.Q AND Alm THEN
	STTimedata[system.stTime.wDay].AlmTime[system.stTime.wHour]:=STTimedata[system.stTime.wDay].AlmTime[system.stTime.wHour]+1;
END_IF

IF STTimedata[system.stTime.wDay].AlmTime[system.stTime.wHour]> 3600 THEN
	STTimedata[system.stTime.wDay].AlmTime[system.stTime.wHour]:= 3600 ;
END_IF

//IF STTimedata[system.stTime.wDay].RunTime[system.stTime.wHour]= 0 AND STTimedata[system.stTime.wDay].WaitTime[system.stTime.wHour]= 0  AND 
  //  (STTimedata[system.stTime.wDay].RunTime[system.stTime.wHour]= 3585  OR  STTimedata[system.stTime.wDay].RunTime[system.stTime.wHour]= 3586 )  THEN
//	STTimedata[system.stTime.wDay].AlmTime[system.stTime.wHour]:= 3600 ;
//END_IF

////////////////换隔膜时间///////////////
rGM_change(CLK:=J , Q=> );

IF rGM_change.Q AND GM_change THEN
	STTimedata[system.stTime.wDay].GMchangeTime[system.stTime.wHour]:=STTimedata[system.stTime.wDay].GMchangeTime[system.stTime.wHour]+1;
END_IF

////////////////剔对齐度时间///////////////
rOverhang_NG(CLK:=J , Q=> );

IF rOverhang_NG.Q AND Overhang_NG THEN
	STTimedata[system.stTime.wDay].OverhangNGTime[system.stTime.wHour]:=STTimedata[system.stTime.wDay].OverhangNGTime[system.stTime.wHour]+1;
END_IF

//数据查询
IF Query THEN
	delay:=TRUE;
END_IF

TON_1(IN:= , PT:=T#60S , Q=> , ET=> );
IF delay THEN
		  IF NOT TON_1.Q THEN
			  TON_1.IN:=TRUE;
		  ELSE	
			  delay:=FALSE;
			  date1:=system.stTime.wDay;
		  END_IF	 
ELSE	
	 TON_1.IN:=FALSE;
END_IF


IF NOT delay THEN
STTimedata[32]:=STTimedata[system.stTime.wDay];
ELSE
STTimedata[32]:=STTimedata[date1];
END_IF

IF (system.stTime.wMonth=2 AND  system.stTime.wDay=28 )   OR
    ((system.stTime.wMonth=4 OR system.stTime.wMonth=6 OR system.stTime.wMonth=9 OR system.stTime.wMonth=11) AND system.stTime.wDay=30 )   OR
	((system.stTime.wMonth=1 OR  system.stTime.wMonth=3 OR system.stTime.wMonth=5 OR system.stTime.wMonth=7 OR system.stTime.wMonth=8 OR system.stTime.wMonth=10 OR system.stTime.wMonth=12) AND  system.stTime.wDay=31)  AND
    system.stTime.wHour=23 AND    system.stTime.wMinute =59 AND   system.stTime.wSecond=59 THEN
	FOR i:=0 TO 32  DO
	MEMSET(ADR(STTimedata[i]),0,SIZEOF(STTimedata[i]));	
	END_FOR
END_IF

END_FUNCTION_BLOCK

// ---- P2POUs/BasicFunction/11_SystemInfo/SystemInfoCtrl.TcPOU
FUNCTION_BLOCK SystemInfoCtrl
VAR_INPUT
	Reset					: BOOL;
	RTCSyncCylce		:	DWORD := 5; (* in seconds *)
	TimeStampTrig		:	BOOL;
END_VAR
VAR_OUTPUT
//	RunTimeNo			: BYTE;
//	ProjectName			: STRING(32);
//	NumberOfTasks		: BYTE;
//	OnlineChangeCount	: UINT;
	RetainVarErr		: BOOL;
	PersistenVarErr	: BOOL;
	TimeStampDT			:	DATE_AND_TIME;
	TimeStamp			:	STRING(25); (* DD.MM.YY-Stunde:Minute:Sekunde:xxx *)
	TimeStr				:	STRING(15);	(* hh.mm.ss.xxms *)
	DateStr				:	STRING(15);	(* dd.mm.jj *)
	TimeStamp2			:	STRING(25); (* YYYY-MM-DD_HHMMSS for example YYYY-MM-DD_HHMMSS_Name.txt *)
	TimeStruct			:	TIMESTRUCT;
	MonthDays			:	WORD;
	LeapYear				:	BOOL;
	WeekOfYear			:	WORD;
	timezoneId			: 	E_TimeZoneID;
END_VAR

VAR
	(* Inst. Get Taskindex *)
	InstGETCURTASKINDEX	: 	GETCURTASKINDEX;
	InstLocalSystemTime	:	FB_LocalSystemTime;

	(* Info: SystemInfo.bootDataFlags
	Bit
	0 RETAIN Variablen: LOADED (fehlerfrei geladen)
	1 RETAIN Variablen: INVALID (es wurde die Sicherungskopie geladen, weil keine g黮tige Datei vorhanden war)
	2 RETAIN Variablen: REQUESTED (RETAIN Variablen sollten geladen werden, Einstellung im TwinCAT System Control))
	3 reserviert
	4 PERSISTENT Variablen: LOADED (fehlerfrei geladen)
	5 PERSISTENT Variablen: INVALID (es wurde die Sicherungskopie geladen, weil keine g黮tige Datei vorhanden war)
	6 reserviert
	7 reserviert *)

	RetainVarLoaded			: BOOL;
	RetainVarInvalid		: BOOL;
	RetainVarRequested		: BOOL;
	PersistentVarLoaded		: BOOL;
	PersistentVarInvalid	: BOOL;

	(* Info: SystemTaskInfoArr	(* Ist ein Array von 1-4 *)
	active					:	BOOL; 		(* Diese Variable zeigt an, ob die Task aktiv ist.*)
	taskName					:	STRING(16);	(* Der Taskname.*)
	firstCycle				:	BOOL;			(* Diese Variable hat im ersten Zyklus der SPS-Task den Wert: TRUE.*)
	cycleTimeExceeded		:	BOOL;			(* In dieser Variablen wird ein 躡erschreiten der eingestellten Taskzykluszeit gemeldet*)
	cycleTime				:	UDINT;		(* Eingestellte Taskzykluszeit in Vielfachen von 100ns*)
	lastExecTime			:	UDINT;		(* Ben鰐igte Zykluszeit f黵 den letzten Zyklus in Vielfachen von 100 ns*)
	priority					:	BYTE;			(* Eingestellte Prioritaet der Task*)
	cycleCount				: 	UDINT;		(* Zykluszaehler*) *)
	_sec						:	WORD;
//	_hour						:	WORD;
END_VAR

(* Get Current Task Index ************************************************************************)
	InstGETCURTASKINDEX();

(* Read System Info Current Task *****************************************************************)
	(* Task Info *)
//	RunTimeNo				:=  _AppInfo.runTimeNo;
//	ProjectName				:=  _AppInfo.ProjectName;
//	NumberOfTasks 			:=  _AppInfo.TaskCnt;
//	OnlineChangeCount		:=  _AppInfo.OnlineChangeCnt;

	(* System Boot Flags *)
//	RetainVarLoaded		:= SystemInfo.bootDataFlags.0;
//	RetainVarInvalid		:= SystemInfo.bootDataFlags.1 ;
//	RetainVarRequested 	:= SystemInfo.bootDataFlags.2 ;
//	PersistentVarLoaded	:= SystemInfo.bootDataFlags.4;
//	PersistentVarInvalid	:= SystemInfo.bootDataFlags.5;


	(* Retein/Persisten Data Err *)
	IF  _TaskInfo[InstGETCURTASKINDEX.Index].FirstCycle THEN
		RetainVarErr		:= NOT RetainVarLoaded AND RetainVarRequested OR RetainVarInvalid;
		PersistenVarErr	:= NOT PersistentVarLoaded OR PersistentVarInvalid;
	ELSIF Reset THEN
		M_Reset();
	ELSE
		;
	END_IF

(* Systemzeit auslesen ************************************************************************)
	InstLocalSystemTime(
		sNetID		:= '',
		bEnable		:= TRUE,
		dwCycle		:= RTCSyncCylce,
		dwOpt			:= (* Default *),
		tTimeout		:= (* Default *),
		bValid		=> ,
		systemTime	=> TimeStruct,
		tzID			=> timezoneId);

	IF TimeStampTrig
		AND InstLocalSystemTime.bValid
	THEN
		(* Date dd.mm.jj ********************)
		IF TimeStruct.wDay < 10 THEN
			DateStr := CONCAT('0',WORD_TO_STRING(TimeStruct.wDay));
		ELSE
			DateStr := WORD_TO_STRING(TimeStruct.wDay);
		END_IF
		DateStr := CONCAT(DateStr,'.');
		IF TimeStruct.wMonth < 10 THEN
			DateStr := CONCAT(DateStr,CONCAT('0',WORD_TO_STRING(TimeStruct.wMonth)));
		ELSE
			DateStr := CONCAT(DateStr,WORD_TO_STRING(TimeStruct.wMonth));
		END_IF
		DateStr := CONCAT(DateStr,'.');
		DateStr := CONCAT(DateStr,RIGHT(WORD_TO_STRING(TimeStruct.wYear),2));
	
		(* Time hh.mm.ss.xxms ***************)
		IF TimeStruct.wHour < 10 THEN
			TimeStr := CONCAT('0',WORD_TO_STRING(TimeStruct.wHour));
		ELSE
			TimeStr := WORD_TO_STRING(TimeStruct.wHour);
		END_IF
		TimeStr := CONCAT(TimeStr,':');
		IF TimeStruct.wMinute < 10 THEN
			TimeStr := CONCAT(TimeStr,CONCAT('0',WORD_TO_STRING(TimeStruct.wMinute)));
		ELSE
			TimeStr := CONCAT(TimeStr,WORD_TO_STRING(TimeStruct.wMinute));
		END_IF
		TimeStr := CONCAT(TimeStr,':');
		IF TimeStruct.wSecond < 10 THEN
			TimeStr := CONCAT(TimeStr,CONCAT('0',WORD_TO_STRING(TimeStruct.wSecond)));
		ELSE
			TimeStr := CONCAT(TimeStr,WORD_TO_STRING(TimeStruct.wSecond));
		END_IF
	
		(* TimeStamp Format DE: DD.MM.YY-Stunde:Minute:Sekunde:xxx,*)
		TimeStamp := CONCAT(DateStr,'-');
		TimeStamp := CONCAT(TimeStamp,TimeStr);
		TimeStamp := CONCAT(TimeStamp,':');
		IF TimeStruct.wMilliseconds > 100 THEN
			TimeStamp:=CONCAT(TimeStamp,WORD_TO_STRING(TimeStruct.wMilliseconds));
		ELSIF TimeStruct.wMilliseconds > 10 THEN
			TimeStamp:=CONCAT(CONCAT(TimeStamp,'0'),WORD_TO_STRING(TimeStruct.wMilliseconds));
		ELSE
			TimeStamp:=CONCAT(CONCAT(TimeStamp,'00'),WORD_TO_STRING(TimeStruct.wMilliseconds));
		END_IF
	
		(* Timestamp Format ENG: YYYY-MM-DD-hh:mm:ss.xxx *)
		(* TimeStamp := SYSTEMTIME_TO_STRING(TimeStruct); *)
	
		(* TimeStamp2 FileName YYYY-MM-DD_HHMMSS *)
		IF _sec <> TimeStruct.wSecond THEN
			TimeStamp2 := CONCAT(WORD_TO_STRING(TimeStruct.wYear),'-');
			IF TimeStruct.wMonth < 10 THEN
				TimeStamp2 := CONCAT(TimeStamp2,CONCAT('0',WORD_TO_STRING(TimeStruct.wMonth)));
			ELSE
				TimeStamp2 := CONCAT(TimeStamp2,WORD_TO_STRING(TimeStruct.wMonth));
			END_IF
			TimeStamp2 := CONCAT(TimeStamp2,'-');
			IF TimeStruct.wDay < 10 THEN
				TimeStamp2 := CONCAT(TimeStamp2,CONCAT('0',WORD_TO_STRING(TimeStruct.wDay)));
			ELSE
				TimeStamp2 := CONCAT(TimeStamp2,WORD_TO_STRING(TimeStruct.wDay));
			END_IF
			TimeStamp2 := CONCAT(TimeStamp2,'_');
			IF TimeStruct.wHour < 10 THEN
				TimeStamp2 := CONCAT(TimeStamp2,CONCAT('0',WORD_TO_STRING(TimeStruct.wHour)));
			ELSE
				TimeStamp2 := CONCAT(TimeStamp2,WORD_TO_STRING(TimeStruct.wHour));
			END_IF
			IF TimeStruct.wMinute < 10 THEN
				TimeStamp2 := CONCAT(TimeStamp2,CONCAT('0',WORD_TO_STRING(TimeStruct.wMinute)));
			ELSE
				TimeStamp2 := CONCAT(TimeStamp2,WORD_TO_STRING(TimeStruct.wMinute));
			END_IF
			IF TimeStruct.wSecond < 10 THEN
				TimeStamp2 := CONCAT(TimeStamp2,CONCAT('0',WORD_TO_STRING(TimeStruct.wSecond)));
			ELSE
				TimeStamp2 := CONCAT(TimeStamp2,WORD_TO_STRING(TimeStruct.wSecond));
			END_IF
			_sec := TimeStruct.wSecond;
	
			(* Jahresinformationen *)
			TimeStampDT := SYSTEMTIME_TO_DT(TimeStruct);
			MonthDays	:= F_GetMaxMonthDays(TimeStruct.wYear,TimeStruct.wMonth);
			LeapYear		:= F_YearIsLeapYear(TimeStruct.wYear) ;
			WeekOfYear	:= F_GetWeekOfTheYear(TimeStampDT);
	
		END_IF
	END_IF

(**************************************************************************************************)

ACTION M_Reset:
RetainVarErr := PersistenVarErr := FALSE;
END_ACTION

END_FUNCTION_BLOCK

// ---- P2POUs/POUS/P2Program_FB.TcPOU
FUNCTION_BLOCK P2Program_FB
VAR_INPUT
	DTselect  :INT;//1、叠台1    2、叠台2    3、叠台3
END_VAR
VAR_OUTPUT
	iTargetTorqueTest:INT;
END_VAR
VAR_IN_OUT
	Sys_Control:System_Control;//系统控制信号
	Mach_Control:ControlSignal;//机架控制信号
	arrCyNo:EleControlNo;//电磙阀控制信号
	AxiseNo:P2_AxiseNo;//轴号
    	TableNo:P2_TableNo;
	CCD:ST_CCDCom;//CCD对接信号
	Par:Parameters;//参数
	Torque:ST_Torque;
END_VAR
VAR
	bFirstFoldFinish:ARRAY[1..5] OF BOOL;//首层隔膜空叠完成  1:首层空叠完成		2：正常电芯空叠完成		3：接带、黄标空叠完成
	iEmptyFoldStep:ARRAY[1..5] OF UINT;//空叠自动步	1:首层空叠	自动步	2：正常电芯空叠自动步	3：接带、黄标自动步
	bEmptyFoldMark:ARRAY[1..5] OF BOOL;//空叠进入流程标志	1:首层空叠	进入流程标志	2：正常电芯空叠进入流程标志	3：接带、黄标进入流程标志

	//fbTensionGM: FB_TensionGMV3;
//新增	
	PosErrorMark: BOOL;//
	AnPosError:ARRAY[1..10] OF BOOL;
	CaPosError:ARRAY[1..10] OF BOOL;
	DTPosError:ARRAY[1..20] OF BOOL;
	
	fActPos:ARRAY [1..20] OF REAL;//轴当前位置
	fSetPos:ARRAY [1..20] OF REAL;//轴当前位置	
	
	
	rDtUse:ARRAY[1..10] OF R_TRIG;//叠台上升沿
	rAnUse:ARRAY[1..10] OF R_TRIG;//正极上升沿
	rCaUse:ARRAY[1..10] OF R_TRIG;//负极上升沿
	fDtUse:ARRAY[1..10] OF F_TRIG;//叠台下降沿
	fAnUse:ARRAY[1..10] OF F_TRIG;//正极下降沿
	fCaUse:ARRAY[1..10] OF F_TRIG;//负极下降沿
	
	tDtUse:ARRAY[1..10] OF TON;//叠台定时器
	tAnUse:ARRAY[1..10] OF TON;//正极定时器
	tCaUse:ARRAY[1..10] OF TON;//负极定时器
	
	fbAnBeltVacuum:FB_Vacuum;//正极模切送料分段皮带1真空
	fbCaMQBeltVacuum:FB_Vacuum;//负极模切送料分段皮带1真空
	fbAnCarryingVacuum:FB_Vacuum;//正极送片搬运升降真空
	fbAndeviationVacuum:FB_Vacuum;//正极纠偏平台真空
	fbAnDTCarryingVacuum:FB_Vacuum;//正极叠片搬运升降真空
	fbCaCarryingVacuum2:FB_Vacuum;//负极送片搬运升降2真空
	fbCaLoadUpBeltVacuum:FB_Vacuum;//负极送片皮带末端真空
	fbCaCarryingVacuum1:FB_Vacuum;//负极送片搬运升降1真空
	fbCadeviationVacuum:FB_Vacuum;//负极纠偏平台真空
	fbCaDTCarryingVacuum	:FB_Vacuum;//负极叠片搬运升降真空

	fbAnCarryingLugVacum: FB_Vacuum;  //正极送片搬运极耳真空
	fbAnDTCarryingLugVacuum: FB_Vacuum; //正极叠片搬运极耳真空
	fbCaCarryingLugVacuum: FB_Vacuum;  //负极送片搬运极耳真空
	fbCaDTCarryingLugVacuum: FB_Vacuum; //负极叠片搬运极耳真空
	fbCaTurnCarryingLugVacuum: FB_Vacuum; //负极送片搬运1旋转极耳真空

	bRectifyRule:ARRAY[1..5] OF BOOL;	//隔膜纠偏条件	
	Ca_deviationFPOKFalg: BOOL;//负极纠偏台是否允许放料
	An_deviationDPOKFalg: BOOL;//正极纠偏台是否允许取料
	An_deviationFPOKFalg: BOOL;//正极纠偏台是否允许放料
	Ca_deviationDPOKFalg: BOOL;//负极纠偏台是否允许取料
	
	
	iMD10: INT;
	iMD11: INT;
	iMD1: INT;//负极
	iND1: INT;//正极----
	iAnCamInSel2: INT;//正极叠片搬运凸轮选择,=1:叠台搬运升降下降取纠偏平台极片
	iAnCamInSel1: INT;//正极送片搬运凸轮选择
	iCaCamInSel1: INT;//负极送片搬运凸轮选择
	iCaCamInSel2: INT;//负极叠片搬运凸轮选择,=1:叠台搬运升降下降取纠偏平台极片
//负极取料过程---判断正极	
	bStandbyStep1_1: BOOL;
	bStandbyStep1_2: BOOL;
//正极取料过程---判断负极	
	bStandbyStep1_3: BOOL;
	bStandbyStep1_4: BOOL;
	
	// 正极取极片初始化步号
	Step_InitAnDT: INT;
	// 负极取片步号
	Step_InitCaDT: INT;
	// 叠片台初始化
	Step_InitDT: INT;
	Step_Init: INT;
	CA_CarryingPos1: BOOL;//负极搬运各轴在取料位，允许凸轮耦合
	CA_CarryingPos2: BOOL;// 判断负极取料机械手的各轴在放料位
	AN_CarryingPos1: BOOL;//正极各轴在取片位
	AN_CarryingPos2: BOOL;//正极各轴在放料位
	arTON: ARRAY[0..15] OF TON;
	Ca_Step0: INT;//负极搬运取流水线极片子程序		
	Ca_Step1: INT;//负极极搬运放极片至纠偏平台
	Ca_Step2: INT;//负极叠片搬运踢料子程序
	Ca_Step3: INT;//负极叠片搬运取纠偏位极片
	Ca_Step4: INT;
	An_Step0: INT;//正极取流水线子程序
	An_Step1: INT;//正极送片搬运放片到纠偏台						
	An_Step2: INT;//正极纠偏平台踢NG片子程序
	An_Step3: INT;//正极取纠偏平台子程序
	An_Step4: INT;
	// 叠片自动程序步
	DP_Step0: INT;

	GluingUpDownagree:BOOL;//拉胶升降轴动作允许
	GluingLineagree:BOOL;//侧贴胶平移轴动作允许
	GluingWhirlingagree:BOOL;//侧贴胶旋转轴动作允行
	
	AN_Carryingagree:BOOL;//正极在安全位允许负极叠片
	Ca_Carryingagree:BOOL;//负极在安全位允许正极叠片
	
	// 正极备料中
	An_standbying: BOOL;
	// 负极备料中
	Ca_standbying: BOOL;
	i: INT;
	r_TailCurl_init: R_TRIG;
	f_TailCurl_init: F_TRIG;
	TON_TailCurl: ARRAY[0..9] OF TON;//尾卷程序延时器
	TON_TailCurl1: ARRAY[0..9] OF TON;//尾卷程序延时器
	TON_Sticker: ARRAY[0..9] OF TON;//贴胶程序延时器
	i1: INT;// 贴胶平移需要移动的位置
	i2: INT;// 贴胶旋转轴需要移动的位置
	// 贴胶记数
	i3: INT;
	r_Sticker_init: R_TRIG;
	f_Sticker_init: F_TRIG;
	TJ_Scan_M: R_TRIG;
	scan_Step :UINT;
	// 隔膜纠偏模拟量值转换
	Rectifydev_V1: Rectifydev_PID;
	TailCultOffloading: INT;
	// 叠台蓝胶检测自动
	DT_BlueGlue: FB_BlueGlue;
	Ca_Demarcate: FB_Demarcate;
	// 负极纠偏自动
	Ca_RecdevPla: FB_RecdevPla;
	// 正极标定自动
	An_Demarcate: FB_Demarcate;
	// 正极纠偏自动
	An_RecdevPla: FB_RecdevPla;

///////////////////////////////////////隔膜缓存/////////////////////////////////////////////////////
   fbGMLengthV1_R  :FB_GMLengthDown_R;
 //  fbGMLengthV2_R  : FB_GMLengthUp_R;
       fbGMLengthV2_R  : FB_GMLengthUp;
   fbGMLengthV1_L  :FB_GMLengthDown_L;
 //  fbGMLengthV2_L  : FB_GMLengthUp_L;
 fbGMLengthV2_L  : FB_GMLengthUp;
	iSetp1: INT;
	fInterval: REAL;

	I10: INT;
	fTagatPos: REAL;
	iNumberOfPoint: INT;
	bExecute: BOOL;

	bExecute2: BOOL;
	bExecute3: BOOL;
	bExecute4: BOOL;
	fTagatPos2: REAL;
	iSetp2: INT;
	I12: INT;
	fInterval2: REAL;
	fJumpPos: REAL;
	fradii: REAL:=12.25;
    fcompensationPos :REAL    :=0.5;
	k_Comp: REAL;

 fbReadCamSlavePos :Tc2_MC2_Camming.MC_ReadCamTableSlaveDynamics;


     arrGMLengthDown_R:  ARRAY[0..3600]  OF REAL;
     arrGMLengthUp_R:  ARRAY[0..3600]  OF REAL;
     arrfTagatPos_R:  ARRAY[0..3600]  OF REAL;
     arrDeltaGMLength_R:  ARRAY[0..3600,0..1]  OF LREAL;  
 


     arrGMLengthDown_L:  ARRAY[0..3600]  OF REAL;
     arrGMLengthUp_L:  ARRAY[0..3600]  OF REAL;
     arrfTagatPos_L:  ARRAY[0..3600]  OF REAL;
    arrDeltaGMLength_L: ARRAY[0..3600,0..1]  OF LREAL;  
    arrDeltaGMLengthAbs_L: ARRAY[0..3600,0..1]  OF LREAL;  
   	fMaxPos: REAL;
	fMinPos: REAL;

        fbCreatCamGMBuffer_R         :FB_CreatCamGMBuffer;
        fbCreatCamGMBuffer_L         :FB_CreatCamGMBuffer;
       fbCreatCamVirGMDriver        :FB_CreatCamVirGMDriver;
       fbCreatCamGMDanserMove         :FB_CrectCamGMDanserMove;

    	iTableSel: INT;

       fbCamInVirGMDriver         :FB_CamIn ;     //放卷虚轴
       fbCamInGMDanserMove   :FB_CamIn ;     //隔膜平移
       fbCamInGMBuffer            :FB_CamIn ;     //隔膜缓存


////////////////////////////////////尾卷/////////////////////////////////////////////////////



	   fbRoll_New  :Dp_Roll_New;//-------------------尾卷正转
	//fbRoll_New  :Dp_Roll_V2;//-----------------------尾卷反转
	
	I20: UINT;
    arrDeltaXmm:   ARRAY[0..3600,0..1]  OF LREAL;  
    arrDeltaYmm:   ARRAY[0..3600,0..1]  OF LREAL;  


	iEndWindCam: INT;
	fMaxPosEndWind: REAL;
	fMinPosEndWind: REAL;
	iNumberOfPointEndWind: UINT;
	fIntervalEndWind: LREAL;
	bEndWindCamDataEnable: BOOL;
    fbCreatCamEndWindX                    :FB_CreatCamEndWind;
    fbCreatCamEndWindY                    :FB_CreatCamEndWind;
    fbCamInEndWindX         :FB_CamIn ;     
    fbCamInEndWindY         :FB_CamIn ;     

	arrGMWindDriverTableData: INT;
	DA2: REAL;
	fAngleRel: REAL;
	GluebHaveTON:TON;

(***************************凸轮表**********************************)
  //负极
      fbCaCrectCamCarryingLine1              :FB_CrectCamMove ;
      fbCaCrectCamCarryingUpDown1       :FB_CrectCamUpDown ;
	  fbCaCrectCamCarryingUpDown1_1	:FB_CrectCamUpDown ;
	  fbCaCrectCamCarryingWhirling			:FB_CrectCamMove;
      fbCaCrectCamCarryingLine2             :FB_CrectCamMove ;
      fbCaCrectCamCarryingUpDown2       :FB_CrectCamUpDown ;
	  fbCaCrectCamCarryingUpDown2_1       :FB_CrectCamUpDown_1 ;
	   fbCaCrectCamCarryingUpDown2_3       :FB_CrectCamUpDown_10 ;
	   
      fbCaCrectCamDTCarryingLine            :FB_CrectCamMove ;
	  
      fbCaCrectCamDTCarryingUpDown     :FB_CrectCamUpDown_3 ;
	  fbCaCrectCamDTCarryingUpDown1     :FB_CrectCamUpDown_2 ;
	  fbCaCrectCamDTCarryingUpDown3     :FB_CrectCamUpDown_10 ;  
      fbCaCamInCarryingLine1                      :FB_CamIn ;    //负极流水线取料平移
      fbCaCamInCarryingUpDown1               :FB_CamIn ;   //负极流水线取料升降
	  fbCaCamInCarryingWhirling                  :FB_CamIn ;   //负极流水线取料旋转
      fbCaCamInCarryingLine2                     :FB_CamIn ;    //负极纠偏平台搬运平移
      fbCaCamInCarryingUpDown2              :FB_CamIn ;    //负极纠偏台搬运平移升降
      fbCaCamInDTCarryingLine                   :FB_CamIn ;    //负极叠台搬运平移
      fbCaCamInDTCarryingUpDown            :FB_CamIn ;    //负极叠台搬运平移升降



//正极
      fbAnCrectCamCarryingLine              :FB_CrectCamMove ;
      fbAnCrectCamCarryingUpDown       :FB_CrectCamUpDown ;
	  fbAnCrectCamCarryingUpDown1       :FB_CrectCamUpDown_1 ;
	  fbAnCrectCamCarryingUpDown3       :FB_CrectCamUpDown_10 ;
	  
	  fbAnCrectCamCarryingWhirling        :FB_CrectCamMove ;	
      fbAnCrectCamDTCarryingLine           :FB_CrectCamMove ;
	  
      fbAnCrectCamDTCarryingUpDown    :FB_CrectCamUpDown_3 ;
	  fbAnCrectCamDTCarryingUpDown1    :FB_CrectCamUpDown_2 ;
	  fbAnCrectCamDTCarryingUpDown3    :FB_CrectCamUpDown_10 ;
	  
      fbAnCamInCarryingLine                     :FB_CamIn ;    //正极纠偏台搬运平移
      fbAnCamInCarryingUpDown              :FB_CamIn ;    //正极纠偏台搬运升降
	  fbAnCamInCarryingWhirling 				 :FB_CamIn ;   //正极纠偏台搬运旋转
      fbAnCamInDTCarryingLine                 :FB_CamIn ;    //正极叠台搬运平移
      fbAnCamInDTCarryingUpDown          :FB_CamIn ;    //正极叠台搬运平移升降

//叠台
     //fbCrectCamLeftYDLine                   :FB_CrectCamYaDaoLine ;   
	fbCrectCamLeftYDLine                   :FB_CrectCamYaDaoLine_V2 ;   
     fbCrectCamLeftYDUpDown             :FB_CrectCamYaDaoUpDown ;
    // fbCrectCamRightYDLine                 :FB_CrectCamYaDaoLine ;
	  fbCrectCamRightYDLine                 :FB_CrectCamYaDaoLine_V2 ;
     fbCrectCamRightYDUpDown           :FB_CrectCamYaDaoUpDown ;

      fbCamInLeftYDLine                       :FB_CamIn ;    //左压刀开合
      fbCamInLeftYDUpDown                :FB_CamIn ;    //左压刀升降
      fbCamInRightYDLine                    :FB_CamIn ;    //右压刀开合
      fbCamInRightYDUpDown             :FB_CamIn ;    //右压刀升降

     // fbCamInVirGM                            :FB_CamIn ;    //拉膜纠偏
      // fbCamInVirGM                            :FB_CamGMVir ;    

      fbGearInGMvir                           :FB_GearInDyn;//--------隔膜纠偏速度模式,,,模式			1：位置模式，，，2：PID模式


	// 负极取料凸轮自动创建程序步
	CaCrectCamStep0: INT;
	// 正极凸轮创建自动程序步
	AnCrectCamStep0: INT;
	// 叠台压刀凸轮自动程序步
	YDCrectCamStep0: INT;
	// 隔膜缓存凸轮自动创建程序步
	GMCreatCamStep0: INT;
	// 尾卷凸轮创建自动程序步
	WZCreatCamStep0: INT;
	// 正极取片凸轮创建
	rCaCreate_TRIG: R_TRIG;
	// 正极取片凸轮创建
	rAnCreate_TRIG: R_TRIG;
	// 叠台压刀凸轮创建
	rYDCreateCam_TRIG: R_TRIG;
	// 隔膜缓存凸轮创建
	rGMCreateCam_TRIG: R_TRIG;
	// 尾卷凸轮创建
	rWZCreateCam_TRIG: R_TRIG;
	// 叠台一键解耦上升沿
	rDTCamOut_TRIG: R_TRIG;	
		// 尾卷一键解耦上升沿
	rWJCamOut_TRIG: R_TRIG;	
	// 负极报警延时
	Ca_AlarmTON: ARRAY[0..19] OF TON;
	// 正极搬运报警时间
	An_AlarmTon:  ARRAY[0..19] OF TON;
	//叠台报警延时
	DT_AlarmTon:  ARRAY[0..19] OF TON;
	//贴胶报警延时
	TJ_AlarmTon:  ARRAY[0..29] OF TON;
	TJ_Error :BOOL;//贴胶真空报警
	// 叠台单步中
	DP_SinStepe: BOOL;
	// 叠台部分凸轮解除耦合
	DP_Step1: INT;
	// 叠片部分轴在耦合中
	DT_AxiseCoupling: BOOL;
	// 叠台主轴启动
	DT_PTP: FB_CamPTPTestV2;
	// 叠台主虚轴启动
	//DT_VriMainExecute: BOOL;


	// 叠台凸轮耦合子程序步
	DP_Step2: INT;
	// 尾卷夹隔膜轴在安全位，允许负极叠片搬运平移至叠片位
	TailCurlSEPTA_SafePos: BOOL;

	// 尾卷单步模式
	TailCurlSinStep: BOOL;
	// 尾卷部分凸轮解除耦合
	TailCurl_Step1: INT;
	// 尾卷拉膜主轴放卷
	tailCult_GearInMultiMaster: MC_GearInMultiMaster;
	// 尾卷放卷虚轴解除耦合
	tailCurl_CamOut: MC_CamOut;
	// 尾卷放卷虚轴下降升沿
	fTailCurl_TRIG: F_TRIG;
	// 夹电芯平移与夹隔膜平移电子齿轮耦合
	//tailCurl_GearIn: MC_GearIn;
	
	tailCurl_GearIn: FB_GearInDyn;//夹电芯平移与夹膜平移电子齿轮
	tailCurl_GearIn1: FB_GearInDyn;//夹电芯平移与夹膜平移电子齿轮---取料
	tailRetGearIn: FB_GearInDyn;//夹电芯平移与夹电芯伸缩电子齿轮
	
	//夹隔膜轴解除耦合
	tailCurl1_CamOut: MC_CamOut;
	//夹隔膜轴下降沿
	fTailCurl1_TRIG: F_TRIG;
	// 尾卷主轴清零自动子程序步
	TailCurlStep0: INT;
	// 尾卷部分轴在耦合中
	TailCurl_AxiseCoupling: BOOL;
	// 尾卷轴在耦合中
	TailCurlCoupling: BOOL;
	// 尾卷长卷针齿轮耦合
	tailCurl1_GearIn: MC_GearIn;
	// 尾卷智短卷针齿轮耦合
	tailCurl2_GearIn: MC_GearIn;
	//尾卷长卷针解除耦合
	tailCurl2_CamOut: MC_CamOut;
	//尾卷短卷针解除耦合
	tailCurl3_CamOut: MC_CamOut;	
	fTailCurl3_TRIG: F_TRIG;
	fTailCurl2_TRIG: F_TRIG;
	// 尾卷轴都在初始位
	TailCurlIinitPos: BOOL;
	// 贴胶单步中
	Sticker_SinStepMode: BOOL;
	// 二维码胶扫码自动程序步
	Stick_Step0: INT;
	// 贴胶子程序
	Stick_Step1: INT;
	// 踢NG胶子程序
	Stick_Step2: INT;
	// 贴胶头前进轴，贴胶时有位置
	i4: INT;
	// 贴胶前进轴运动允许
	GluingRetractingagree: BOOL;
	// 正极回原点延时
	An_GohomeTon: TON;
	An_RectifydevGohomeTon: TON;	
	// 负极回原点
	Ca_GohomeTon: TON;
	Ca_RectifydevGohomeTon: TON;		
	// 负极回原点启动上升沿
	rCa_Gohome_TRIG: R_TRIG;
	// 纠偏程序步
	Ca_Demarcate_Step0: INT;
	// 负极纠偏自动程序步
	Ca_RecdevPla_Step0: INT;
	// 正极纠偏标定程序步
	An_Demarcate_Step0: INT;
	// 正极纠偏定位程序步
	An_RecdevPla_Step0: INT;
	// 正极取片回原点上升沿
	rAn_Gohome_TRIG: R_TRIG;
	// 正极取片回原点下降沿
	fAn_Gohome_FRIG: Tc2_Standard.F_TRIG;
	// 叠台回原点启动上升沿
	rDT_GohmeTRGI: R_TRIG;
	// 叠台回原点启动下降沿
	fDT_GohmeTRGI: Tc2_Standard.F_TRIG;
	// 叠片回原点上升沿启动
	r_DTinitiStart: R_TRIG;
	f_DTinitiStart: R_TRIG;
	Ca_RectifydevStep: INT;
	// CCD第一次拍照超时报警
	CCD_Ton: TON;
	// 正极CCD标定NG
	rAnCCD_Ton: TON;
	// 正纠偏自动程序步
	An_StandbyStep0: INT;
	rPoleIn_btn: R_TRIG;
	rPoleTapeL_btn: R_TRIG;
	rPoleTapeR_btn: R_TRIG;
	// 叠台已叠极片计数
	rDT_Count: R_TRIG;
//	sFB_TensionGMV2_1: FB_TensionGMV2_1;
	fbTensionGM: FB_TensionGMV3;
      fbRectifyGM:   FB_RectifyGM;


     rtGMMoveCount :       Tc2_Standard.R_TRIG;

	Ca_CanIn1: BOOL;//叠负极片凸轮耦合1
	Ca_CanIn2:BOOL;//叠负极片凸轮耦合2
	Ca_CanIn3: BOOL;//叠负极片凸轮耦合3
	Ca_CanIn4:BOOL;//叠负极片凸轮耦合4	
	
	An_CanIn1: BOOL;//叠正极片凸轮耦合1
	An_CanIn2:BOOL;//叠正极片凸轮耦合2
	An_CanIn3: BOOL;//叠正极片凸轮耦合3
	An_CanIn4:BOOL;//叠正极片凸轮耦合4	
	fbGearInGMvirbEnable: BOOL;
	// 单步启动上升沿
	rDT_SinStepd: R_TRIG;
	// 取负极片自动程序步
	Ca_StandbyStep0: INT;
	// 取正极片自动程序步
	An_StandbyStep1: INT;
	// 负极报警复位上升沿
	rCa_AlarmReset: R_TRIG;
	// 负极报警复位下降沿
	fCa_AlarmRest: F_TRIG;
	// 负极取料皮带自动程序步
	Ca_StandbyStep2: INT;
	// 正极取片报警复位上升沿
	rAn_AlarmRest: R_TRIG;
	// 正极取片报警复位下降沿
	fAn_AlarmRest: F_TRIG;
	// 叠片台报警复位上升沿
	rDT_AlarmRest: R_TRIG;
	// 叠台报警复位下降沿
	fDT_AlarmRest: F_TRIG;
	// 负极流水线延时间
	Ca_BeltTon: TON;
	// 正极流水线取料完成复位时间
	An_BeltTon: TON;
	Ca_StandbyStep3: INT;
	// 负极取流水线各轴在取片初始位
	CaCarryingPos1: BOOL;
	// 负极取流水线极片各轴在放片位
	CaCarryingPos2: BOOL;
	// 负极缓存流水线程序步
	Ca_StandbyStep4: INT;
	// 耦合中的轴报警
	arrAxisCamError: BOOL;
	// 叠片耦合中的轴报警停止主轴
	rArrAxisCamError: R_TRIG;
	rCodeGluePressCy_btn: R_TRIG;
	rGluePressCy_btn: R_TRIG;
	// 叠台真空、破真空、取片条件
	DP_Step3: INT;

	An_StandbyStep2: INT;	// 正极主轴凸轮真空、破真空、标记位
	Ca_StandbyStep1: INT;	// 正极主轴凸轮真空、破真空、标记位
	// 一键张力启动
	rTension_Start: R_TRIG;
	// 一键备蓝胶按钮启动
	rStickerStandbyBule_btn: R_TRIG;
	// 一键备二维码胶按钮启动
	rStickerStandbyCode_btn: R_TRIG;
	// 贴胶程序步1
	Sticker_Step0: INT;
	Sticker_Step1: INT;
	Sticker_Step2: INT;
	// 贴胶程序步2
	fStickerStandbyCode_btn: F_TRIG;
	fStickerStandbyBule_btn: F_TRIG;
	StandbyCode_Start: BOOL;
	StandbyBule_Start: BOOL;
	rStickerStart_HMI: R_TRIG;

    csCodeTcp:CS_CodeTcp;
    iCode2: ICode;
	SlaveOffset: LREAL := 0;
	tDT_GohomeTON: TON;
	// 判断叠台主轴是否完成步序
	DP_Step4: INT;//叠台下降
	DP_Step5: INT;//正负极运动过程中真空判断
	DP_Step6: INT;//正极数据绑定
	DP_Step7: INT;//负极数据绑定
	
	// 一键初始化步
	AllGohomeStep: INT;	
	AllGohome_Hbtn :BOOL;//一键初始化，触摸屏按钮
	AllGohome_Done:BOOL;//一键初始化完成
	r_AllGohome: R_TRIG;
	f_AllGohome: F_TRIG;
	AllGohomeTon:ARRAY[1..10] OF Tc2_Standard.TON;
	// 尾卷初始化步
	TailCurlStep1: INT;
	// 尾卷回原点步
	tTailCurlTON: TON;
	// 夹膜平移轴动作允许
	TailCurlSEPTALineGoargee: BOOL;
	// 单步启动上升沿
	rWJ_SinStepd: R_TRIG;
	// 贴胶回原点步
	StickerStep0: INT;
	tStickerTON: TON;
	// 破真空时间
	pt_Time: TIME;
	Ca_BeltGohomeTon: TON;
	rCa_BeltGohome_TRIG: R_TRIG;
	Step_InitCaDT0: INT;
	esle: INT;
	
	Ca_StandbyStep5: INT;// 判断主轴是否完成
	// 判断正极主轴是否完成
	An_StandbyStep3: INT;
	An_CamTON: TON;
	rClearcountR_TRIG: R_TRIG;
	fCa_Gohome_TRIG: F_TRIG;
	fCa_BeltGohome_TRIG: F_TRIG;


	tCaCreate_TON: TON;
	tYDCreateCamTON: TON;
	tGMCreateCamTON: TON;
	tWZCreateCamTON: TON;
	SLCurlingneedleLine_TON :TON;//转针旋转回初始位延时
	AG: BOOL;
	tailCurlGearInEnable: BOOL;
	tailRetGearInEnable: BOOL;
	tailCurlGearInEnable1: BOOL;//取料
	// 负极CCD拍照完成
	Ca_CCD_Done: BOOL;
	rCa_RecdevPlaR_TRIG: R_TRIG;
	An_CCD_Done: BOOL;
	rAn_RecdevPlaR_TRIG: R_TRIG;
	AV: BOOL;
	tMach_Control_TON: TON;
	avg: BOOL;
	TailCurlStep3: INT;
	TailCurlStep4: INT;
	TailCurlStep6: INT;
	TailCurlStart: BOOL;
	fbAnCamInCarryingUpDownOutCam_F_TRIG: F_TRIG;
	// 正极搬运升降凸轮解耦标记
	fbAnCamInCarryingUpDownOutCamFlge: BOOL;
	fbAnCamInCarryingUpDownOutCam1_F_TRIG: F_TRIG;
	fbCaCamInCarryingUpDown2OutCam_F_TRIG: F_TRIG;
	//fbCaCamInCarryingUpDown2OutCamFlge: BOOL;//负极升降2凸轮解耦标记	
	fbCaCamInCarryingUpDown2OutCam1_F_TRIG: F_TRIG;
	An_NG_TON: TON;
	An_NG_TON2: TON;
	avg1: BOOL;
	Ca_NG_TON: TON;
	Ca_NG_TON2: TON;
	test1:BOOL;
	StickerGohome_TON  :ARRAY[1..30] OF Tc2_Standard.TON;
	Scan_TON		   :ARRAY[1..30] OF Tc2_Standard.TON;//叠台用延时
	WJ_TON :ARRAY[1..30] OF Tc2_Standard.TON;
	Ca_TON :ARRAY[1..30] OF Tc2_Standard.TON;
	An_TON :ARRAY[1..30] OF Tc2_Standard.TON;
	DT_Home_TON :ARRAY[1..30] OF Tc2_Standard.TON ;
	Ca_Cam_ton :ARRAY[1..30] OF Tc2_Standard.TON;
	An_Cam_ton :ARRAY[1..30] OF Tc2_Standard.TON;
	DT_Cam_ton :ARRAY[1..30] OF Tc2_Standard.TON;
	WJ_Cam_ton :ARRAY[1..30] OF Tc2_Standard.TON;
	stTime		:TIMESTRUCT;
	NT_GetTime1: NT_GetTime;
	strTime: STRING;
	fbLON:BOOL;
	//fbLON: R_TRIG;
	fbLOFF: BOOL;
	fbComOpen: BOOL;
	fbComClose: BOOL;
	//bCS_CodeTcp: CS_CodeTcp;
	TON_2: Ton;
	fbinit_tcp: BOOL;
	IP_A: T_IPv4Addr;

	x1: LREAL;
	x2: LREAL;
	y: LREAL;
	q1: INT;
	// 负极取极片回原点完成
	Ca_GohomeDone: BOOL;
	// 负极取极片回原点中
	Ca_Gohoming: BOOL;
	// 负极皮带初始化完成
	Ca_BeltGohomeDone: BOOL;
	// 负极皮带回原点中
	Ca_BeltGohoming: BOOL;
	Ca_GohomeOverTon: TON;
	Ca_BeltGohomeOverTon: TON;
	TailCurlStep5: INT;
	An_GohomeDone: BOOL;// 正极取极片回原点完成
	WZIniti_Done: BOOL;

    An_Gohoming: BOOL;// 正极取极片回原点中
    An_GohomeOverTon: TON;// 正极取极片回原点延时
    
    Dietai_GohomeDone: BOOL;// 叠台回原点完成 
	Dietai_Gohoming: BOOL;// 叠台回原点中
	Dietai_GohomeOverTon: TON;// 叠台回原点延时
	
	Tailcurl_GohomeDone: BOOL;// 尾卷回原点完成 
	Tailcurl_Gohoming: BOOL;// 尾卷回原点中
	Tailcurl_GohomeOverTon: TON;//尾卷回原点延时
	
	Sticker_GohomeDone: BOOL;// 贴胶回原点完成 
	Sticker_Gohoming: BOOL;// 贴胶回原点中
	Sticker_GohomeOverTon: TON;//尾贴回原点延时
	
	
	


	rAnCCD_Ton1: TON;
	An_CQ_ton :Tc2_Standard.TON;
	Ca_CQ_ton :Tc2_Standard.TON;
	CCD_Ton1: TON;
	GluingUpDownPoint1: REAL;
	rMarkesensorR_TRIG: R_TRIG;
	GluingUpDownPoint2: REAL;
	GluingUpDownPoint3: REAL;
	GluingUpDownPoint4: REAL;
	
	// CCD心跳异常
	CDD_HeartTON1: TON;
	CDD_HeartTON2: TON;
	rTailCurl_AlarmRest: R_TRIG;
	fTailCurl_AlarmRest: F_TRIG;
	rSticker_AlarmRest: R_TRIG;
	fTSticker_AlarmRest: F_TRIG;
	DTIniti_Done: BOOL;
	TJIniti_Done: BOOL;
	
	//CCD通讯测试
	rtAn_CCDTest1:R_TRIG;
	rtAn_CCDTest2:R_TRIG;
	rtAn_CCDTest3:R_TRIG;
	rtAn_CCDTest4:R_TRIG;
	tonAn_CCDTest1:TON;
	tonAn_CCDTest2:TON;
	bAn_CCDTest1:BOOL;
	bAn_CCDTest2:BOOL;
	
	rtCa_CCDTest1:R_TRIG;
	rtCa_CCDTest2:R_TRIG;
	rtCa_CCDTest3:R_TRIG;
	rtCa_CCDTest4:R_TRIG;
	tonCa_CCDTest1:TON;
	tonCa_CCDTest2:TON;
	bCa_CCDTest1:BOOL;
	bCa_CCDTest2:BOOL;		
	// 主轴启动超时报警延时
	VirMain_TON: TON;
	CurlingneedleLine_GearIn: FB_GearInDyn;
	// 长、短卷针平移电子齿轮耦合启动
	CurlingneedleLineEnable: BOOL;
	CamOutArgel: REAL;
	//主轴定位时间t
	VirMain_TagatTime:REAL;
	Ca_Number: BOOL;
	An_Number: BOOL;
	An_NG :INT;
	Ca_NG :INT;
	An_NGTest1:R_TRIG;
	Ca_NGTest1:R_TRIG;
	Pole_BJ: BOOL;
	An_StandbySub3_ton :ARRAY[1..6] OF Tc2_Standard.TON ;
	Ca_StandbySub3_ton :ARRAY[1..6] OF Tc2_Standard.TON ;
	NN :INT;//对齐度NG计数
	D :UINT;
	An_dppy_Xzb:REAL;//正极叠片平移轴X坐标位置
	Ca_dppy_Xzb:REAL;//负极叠片平移轴X坐标位置	
	TailCurl_WJJMPY_Xzb:REAL;//尾卷夹膜平移轴X坐标位置
	
	AnAxisbstop_R: R_TRIG;
	AnAxisbstop_F: F_TRIG;
	CaAxisbstop_R: R_TRIG;
	CaAxisbstop_F: F_TRIG;
	
	AnAxisbstop1_R: R_TRIG;
	AnAxisbstop1_F: F_TRIG;
	CaAxisbstop1_R: R_TRIG;
	CaAxisbstop1_F: F_TRIG;
	
	TailCurlAxisbstop_R: R_TRIG;
    TailCurlAxisbstop_F: F_TRIG;
	
	AnError_r: R_TRIG;
	CaError_r: R_TRIG;
	WJError_r: R_TRIG;
	
	DayClear1:R_TRIG;
	NightClear1:R_TRIG;
	
	rOverhangNG:R_TRIG;
	
//力矩判断标志位
	An_CarryingTorMark:BOOL:=FALSE;//正极搬运1移位力矩判断标志位
	An_DTCarryingTorMark:BOOL:=FALSE;//正极叠台搬运力矩判断标志位
	Ca_Carrying1TorMark:BOOL:=FALSE;//负极搬运1平移力矩判断标志位
	Ca_Carrying2TorMark:BOOL:=FALSE;//负极搬运2平移力矩判断标志位
	Ca_DTCarryingTorMark:BOOL:=FALSE;//负极叠台搬运平移力矩判断标志位
	TailCurlTorMark:BOOL:=FALSE;//尾卷夹电芯平移力矩判断标志位
	TailCurlWhirlTorMark:BOOL:=FALSE;//尾卷夹电芯旋转力矩判断标志位
	TailCurlSEPTATorMark:BOOL:=FALSE;//夹膜平移力矩判断标志
	//TailCurlRetMark:BOOL:=FALSE;//尾卷夹电芯伸缩力矩判断标志
	DP_Step8: INT;//纠偏平台有无极片复检----运动过程中检测纠偏平台有无片  主轴118-123°
	DP_CaNumber: INT;//叠台放多片检测------DP_Step9-----屏蔽
	DP_AnNumber: INT;//叠台放多片检测------DP_Step9-----屏蔽
	DP_Step9: INT;//连续叠2片正极或者负极防呆检测
	DP_Number_ton: TON;//延时
	//TorqueTime:ARRAY [1..9] OF TON;
	rtFlgGMEndIng: R_TRIG;
	bFlgGMEndIng: BOOL;
	ftFlgGMEndIng: F_TRIG;
	fGMEndSatrtPos: REAL;
	fGMEndLength: REAL;
	Ca_CanIn7: BOOL;
	Ca_CanIn6: BOOL;
	Ca_CanIn5: BOOL;
	An_CanIn7: BOOL;
	An_CanIn6: BOOL;
	An_CanIn5: BOOL;
	DP_CheseCam: BOOL;//叠片结束后空叠隔膜功能开启标记--判断正极取片升降凸轮是否耦合
	
	rtGMBtn: R_TRIG;
	rtGMBtn2: R_TRIG;
	iGMCheckSetp: INT;
	iCa_QuantitedRecord: UINT;
	fGMLengthRecord: REAL;
	bFlgGMPulling: BOOL;
	iWindDiameterRecord1: REAL;
	iWindDiameterRecord2: REAL;
	Ca_CanIn8: BOOL;
	DT_Readydown: BOOL;
	Ca_YS: Ton;
	Ca_YS1: Ton;
	YS: Ton;
	YS1: Ton;
	YS2: Ton;
	TailCurlSplintCy_TON: Ton;
	TailCurlSplintCy_ON: Ton;
	CamOut_TON: TON;
	OFF: INT;
	P2M_BlueFlag: FB_BlueFlag;
	stNumberPos: ARRAY [0..20] OF LREAL;
	stNumberPos1: ARRAY [0..20] OF LREAL;
	stNumberPos2: ARRAY [0..20] OF LREAL;	
	hot_time_ton: Ton;
	
	Bnt_Blueflaging: BOOL;
	DT_Ca_Quantited: UINT;
	Blueflaging: BOOL;
	
	fRectifyTimeAdjust1           :REAL;  //纠偏时间
	BulebntR_TRIG: R_TRIG;//蓝胶接带上升沿
	YellowmarkR_TRIG: R_TRIG;//隔膜色标感应器上升沿
	JumpPiceReady_temp1: BOOL;
	JumpPiceReady_temp2: BOOL;
	JumpPiceReady_temp3: BOOL;
	fbAnCrectCamUpDown_4: FB_CrectCamUpDown_4;
	JumpPiceReady_temp4: BOOL;
	JumpPiceReady_temp5: BOOL;
	iMode: INT;
	
	rAnCCDStart: R_TRIG;
	rCaCCDStart: R_TRIG;
	AnCCDMark: BOOL;//正极CCD拍照标志
	CaCCDMark: BOOL;//负极CCD拍照标志
	
	DP_Step11: UINT;    // 正极纠偏平台回原
	DP_Step12: UINT;	// 负极纠偏平台回原
	
	WJ_ET:TIME;//尾卷时间
	An_CCDNG:INT;//正极CCD抛片计数
	Ca_CCDNG:INT;//负极CCD抛片计数
	BlueGlue_JS: INT;
	//fbCadeviationVacuum: INT;
	P2Ca_M: INT;
	Vacuumsel: INT;
	Ca_NGStep: INT;
	//fbAnCarryingVacuum: INT;
	//fbAndeviationVacuum: INT;
	P2An_M: INT;
	Andeviation_date: INT;
	AnCarrying_date: INT;
	
	rtEnable		:R_TRIG;  
	ftEnable		:F_TRIG;
	Test:	BOOL;
	KD_Mark:BOOL;//空叠隔膜中
	DTR_Trig: INT;
	An_JumpRules:ARRAY[1..10] OF BOOL;//正极跳取条件
	Ca_JumpRules:ARRAY[1..10] OF BOOL;//正极跳取条件
	
	rtVacuum1: R_TRIG;
	ftVacuum1: F_TRIG;
	rtVacuum2: R_TRIG;
	ftVacuum2: F_TRIG;
	rtVacuum3: R_TRIG;
	ftVacuum3: F_TRIG;
	
	iTest1:INT;
	rtCCDStart: INT;
	An_Rectifydev_JS: INT;
	
	iTensionAutoStep:UINT;//叠台自动启动时张力自动步
	
	//叠台提速COE寻址修改直线电机参数
	FB_EcCoESdoWrite_SEPTATLine : ARRAY[1..4] OF FB_EcCoESdoWrite;   //隔膜平移参数修改
	FB_EcCoESdoWrite_SEPTATCache : ARRAY[1..4] OF FB_EcCoESdoWrite;	  //隔膜缓存参数修改
	FB_EcCoESdoWrite_AnCarryingLine : ARRAY[1..4] OF FB_EcCoESdoWrite;	  //正极送片搬运平移参数修改
	FB_EcCoESdoWrite_AnDTCarryingLine : ARRAY[1..4] OF FB_EcCoESdoWrite;	  //正极叠片搬运平移参数修改
	FB_EcCoESdoWrite_CaCarryingLine2 : ARRAY[1..4] OF FB_EcCoESdoWrite;  //负极送片搬运平移参数修改
	FB_EcCoESdoWrite_CaDTCarryingLine : ARRAY[1..4] OF FB_EcCoESdoWrite;	  //负极叠片搬运平移参数修改
	
	Rectifydev1:REAL;
	Rectifydev2:REAL;
	
	DPcount:UINT;//叠片计数
	LMcount:UINT;//拉膜计数
	NGcount:UINT;//NG拉膜计数
	DPGMlength:REAL;//单个电芯隔膜长度
	rGMmanual: R_TRIG;
	
	fDiameterORLength: FB_DiameterORLength;
	bDiameterAlarm:BOOL;
	
	//改OH NG踢废运动控制
	bMoveFowerdR: BOOL;
	bMoveFowerdL: BOOL;
	arrfTagatPos2_R:  ARRAY[0..3600]  OF REAL;
	arrDeltaGMLength2_R:  ARRAY[0..3600,0..1]  OF LREAL;  
    arrGMLengthDown2_R:  ARRAY[0..3600]  OF REAL;
	
	arrfTagatPos2_L:  ARRAY[0..3600]  OF REAL;
	arrDeltaGMLength2_L:  ARRAY[0..3600,0..1]  OF LREAL;  
    arrGMLengthDown2_L:  ARRAY[0..3600]  OF REAL;
	arrDeltaGMLength2Abs_L: ARRAY[0..3600,0..1]  OF LREAL;  
	
	 fbCreatCamGMBuffer2_R         :FB_CreatCamGMBuffer;	
	 fbCreatCamGMBuffer2_L         :FB_CreatCamGMBuffer;
	 fbCreatCamVirGMDriver2        :FB_CreatCamVirGMDriver;
	
       fbCamInVirGMDriver2         :FB_CamIn ;    
       fbCamInGMBuffer2            :FB_CamIn ;     
	
	An_OverNGMark:BOOL;//正极片对齐度NG
	Ca_OverNGMark:BOOL;//负极片对齐度NG
	Ca_OverNGStep: INT;//踢负极片对齐度NG
	An_OverNGStep: INT;//踢正极片对齐度NG	
	
	DT_TON:ARRAY[1..6] OF Tc2_Standard.TON ;
	An_OverhangNG:BOOL;//正极片对齐度NG
	Ca_OverhangNG:BOOL;//负极片对齐度NG
	rtVacALM: ARRAY[1..5] OF R_TRIG;
	
	GMlappos  : ARRAY[1..4] OF LREAL;
	AnOverNGcount :INT;//正极片对齐度NG计数
	CaOverNGcount :INT;//负极片对齐度NG计数
	OversequelNG:BOOL;//单片踢废对齐度连续NG
	
	AN_RectifyTry_fb: FB_RectifyTry;
	Ca_RectifyTry_fb: FB_RectifyTry;
    An_SuckerTest_fb:FB_SuckerTest;
	Ca_SuckerTest_fb:FB_SuckerTest;	
	
	//20240415 对齐度闭环
	iCaOverhandCount1_Y: UINT;//满足20片+1计数
	fCaMeanSingle_Y: REAL;//当前片Mean中值
	fCaSUMMean_Y: REAL;//20片周期Mean求和
	iCaOverhandCount2_Y: UINT; //20片周期内有效计算片数
	fCaArvMean_Y: REAL; //20片Mean平均值
	fCaOffsetMean_Y: REAL; //Y方向偏差值 给纠偏台补偿值  下个电芯是否清0？？
	fCaMeanBase_Y: REAL;//基准值
	
		iCaOverhandCount1_X: UINT;//满足20片+1计数
	fCaMeanSingle_X: REAL;//当前片Mean中值
	fCaSUMMean_X: REAL;//20片周期Mean求和
	iCaOverhandCount2_X: UINT; //20片周期内有效计算片数
	fCaArvMean_X: REAL; //20片Mean平均值
	fCaOffsetMean_X: REAL; //Y方向偏差值 给纠偏台补偿值  下个电芯是否清0？？
	fCaMeanBase_X: REAL;//基准值
	
	
	(*
	iAnOverhandCount1: UINT;//满足20片+1计数
	fAnMeanSingle: REAL;//当前片Mean中值
	fAnSUMMean: REAL;//20片周期Mean求和
	iAnOverhandCount2: UINT; //20片周期内有效计算片数
	fAnArvMean: REAL; //20片Mean平均值
	fAnOffsetMean: REAL; //Y方向偏差值 给纠偏台补偿值  下个电芯是否清0？？
	fAnMeanBase: REAL;//基准值
	*)
	
	fAnScaling:REAL:=1;//比例系数 20240508 CF
	fCaScaling:REAL:=1;//比例系数 20240508 CF	
	
	DPtime:INT ;
	DPtime1:INT ;
	//20240521 WCZ
	fbCrectCamLeftYDLine2               :FB_CrectCamYaDaoLine2_V2 ;   
    fbCrectCamLeftYDUpDown2             :FB_CrectCamYaDaoUpDown2 ;	 
	fbCrectCamRightYDLine2              :FB_CrectCamYaDaoLine2_V2;
	fbCrectCamRightYDUpDown2            :FB_CrectCamYaDaoUpDown2 ;

END_VAR

//负极备极片自动程序
Ca_Alarm();//负极报警
Ca_Conditions();//负极安全条件
Ca_Cam();//负极凸轮
Ca_Gohome();//负极回原点
Ca_StandbyMain();//负极备极片主程序
Ca_StandbyMain2();//负极备极片主程序
Ca_StandbySub1();//负极取流水线极片子程序
Ca_StandbySub2();//负极放纠偏极片子程序
Ca_StandbySub3();//负极踢NG料子程序
Ca_StandbySub4();//负极取纠偏极片子程序
Ca_Cahebelt();//负极皮带缓存自动
Ca_Rectifydev();//负极纠偏自动
//Par.iModeEN.DT_CCD_TwoModelEN;
//正椎备极片自动程序
An_Alarm();//正极报警
An_Conditions();//正极安全条件
An_Cam();//正极凸轮
An_Gohome();//正极取片回原点
An_StandbyMain();//正极备极片主程序
An_StandbyMain2();//正极备极片主程序
An_StandbySub1();//正极取流水线极片子程序
An_StandbySub2();//正极放纠偏极片子程序
An_StandbySub3();//正极踢NG料子程序
An_StandbySub4();//正极取纠偏极片子程序
An_Rectifydev();//正极纠偏自动

//叠台自动程序
_01_DT_Product();
DT_Condition();
DT_Alarm();//报警
GMBufferLengthCalculate();//隔膜级存计算
GMBufferCam();//隔膜缓存凸轮生成
Dietai_Cam();//压刀凸轮
Dietai_Gohome();//叠台轴回原点
_01DT_Auto();
_01DT_Auto2();
_01DT_Auto3();
_01DT_Auto4();
_01DT_Auto5();
_01DT_AutoSub1_CamOut();
_02BlueGlue_Auto();
_03Rectifydev_Auto();
_04Tension_Auto();
An_OverNG();
Ca_OverNG();
GMEmptyFold1();
GMEmptyFold2();
GMEmptyFold3();
ModeENLimk();
MotionCoe_Write();
//尾卷自动程序
TailCurl_Alarm();//报警
TailCurl_Condition();//尾卷安全条件
TailCurl_Gohome();//尾卷回原点
TailCurlCam();//尾卷凸轮
TailCurl_Auto1();//尾卷上、下电芯自动
TailCurl_Auto2();//尾卷卷电芯自动
Tailcurl_Auto_CamOut();//尾卷凸轮解耦



//贴胶程序
Sticker_Alarm();//报警
Stick_Condition();//贴胶安全条件
Sticker_Gohome();//贴胶回原点


_01Sticker_Auto();//贴胶自动程序
_02Sticker_Auto();//备胶自动程序
_02Sticker_AutoSbu1_Scan();//二维码胶扫码自动子程序
_02Sticker_AutoSbu2_NG();//二维码胶扫码NG胶踢胶子程序
Code();//二维码Tcp通讯





Manual();
P2_Init();
Vacuum_Signal();

All_GoHome();
TorqueCheckAlarm();
AA1;

ACTION _01_DT_Product:

//电芯数清零
IF Mach_Control.DT_b.DT_amount_clear THEN
	Mach_Control.DT_b.DT_amount:=0;
	Mach_Control.DT_b.DT_amount_clear:=FALSE;
END_IF


//对齐度NG统计
         rOverhangNG(CLK:=Mach_Control.DT_b.Overhang_TF , Q=> );
//白班 踢对齐度NG数/总叠片数		 
(*         IF HMI_Hour>=8 AND HMI_Hour<20 THEN
			 IF rOverhangNG.Q AND NOT  Mach_Control.U.EmptyRunMode AND Mach_Control.DT_b.DT_Oerhang_Z=2 THEN
				Mach_Control.DT_b.DT_DayHough :=Mach_Control.DT_b.DT_DayHough+(UINT_TO_REAL(Par.stDT_date.DT_Overhang_SUM)*2/(UINT_TO_REAL(Par.stDT_date.An_Quantity)+UINT_TO_REAL(Par.stDT_date.Ca_Quantity))); 
				Mach_Control.DT_b.DT_DayHough_U :=Mach_Control.DT_b.DT_DayHough_U+1;
			 END_IF
		 END_IF
		 *)
        IF HMI_Hour>=8 AND HMI_Hour<20 THEN
			 IF rOverhangNG.Q AND NOT  Mach_Control.U.EmptyRunMode AND NOT Blueflaging  THEN
				Mach_Control.DT_b.DT_DayHough :=Mach_Control.DT_b.DT_DayHough+UINT_TO_REAL(Mach_Control.An_b.An_Quantited(*+Mach_Control.Ca_b.Ca_Quantited*))/(UINT_TO_REAL(Par.stDT_date.An_Quantity)(*+UINT_TO_REAL(Par.stDT_date.Ca_Quantity)*)); //JR
				Mach_Control.DT_b.DT_DayHoughAn:=Mach_Control.DT_b.DT_DayHoughAn+UINT_TO_REAL(Mach_Control.An_b.An_Quantited); 
				Mach_Control.DT_b.DT_DayHoughCa:=Mach_Control.DT_b.DT_DayHoughCa+UINT_TO_REAL(Mach_Control.Ca_b.Ca_Quantited); 
				Mach_Control.DT_b.DT_DayHough_U :=Mach_Control.DT_b.DT_DayHough_U+1;
			 END_IF
		 END_IF
        IF HMI_Hour>=8 AND HMI_Hour<20 THEN
			 IF rOverhangNG.Q AND NOT  Mach_Control.U.EmptyRunMode AND Blueflaging  THEN
				Mach_Control.DT_b.DTJD_DayHough :=Mach_Control.DT_b.DTJD_DayHough+UINT_TO_REAL(Mach_Control.An_b.An_Quantited(*+Mach_Control.Ca_b.Ca_Quantited*))/(UINT_TO_REAL(Par.stDT_date.An_Quantity)(*+UINT_TO_REAL(Par.stDT_date.Ca_Quantity)*)); //JR
				Mach_Control.DT_b.DTJD_DayHoughAn:=Mach_Control.DT_b.DTJD_DayHoughAn+UINT_TO_REAL(Mach_Control.An_b.An_Quantited); 
				Mach_Control.DT_b.DTJD_DayHoughCa:=Mach_Control.DT_b.DTJD_DayHoughCa+UINT_TO_REAL(Mach_Control.Ca_b.Ca_Quantited); 
				Mach_Control.DT_b.DTJD_DayHough_U :=Mach_Control.DT_b.DTJD_DayHough_U+1;
			 END_IF
		 END_IF
//晚班 踢对齐度NG数/总叠片数		  
(*		IF ((HMI_Hour>=0 AND HMI_Hour<8) OR  (HMI_Hour>=20 AND HMI_Hour<=23))AND NOT  Mach_Control.U.EmptyRunMode THEN
			 IF rOverhangNG.Q THEN
			   Mach_Control.DT_b.DT_NightHough:=Mach_Control.DT_b.DT_NightHough+(UINT_TO_REAL(Par.stDT_date.DT_Overhang_SUM)*2/(UINT_TO_REAL(Par.stDT_date.An_Quantity)+UINT_TO_REAL(Par.stDT_date.Ca_Quantity)));
               Mach_Control.DT_b.DT_NightHough_U :=Mach_Control.DT_b.DT_NightHough_U+1; 
			 END_IF
		 END_IF 
		 *)
        IF ((HMI_Hour>=0 AND HMI_Hour<8) OR  (HMI_Hour>=20 AND HMI_Hour<=23)) THEN
			 IF rOverhangNG.Q AND NOT  Mach_Control.U.EmptyRunMode AND NOT Blueflaging THEN
				Mach_Control.DT_b.DT_NightHough :=Mach_Control.DT_b.DT_NightHough+UINT_TO_REAL(Mach_Control.An_b.An_Quantited(*+Mach_Control.Ca_b.Ca_Quantited*))/(UINT_TO_REAL(Par.stDT_date.An_Quantity)(*+UINT_TO_REAL(Par.stDT_date.Ca_Quantity)*)); 
				Mach_Control.DT_b.DT_NightHoughAn:=Mach_Control.DT_b.DT_NightHoughAn+UINT_TO_REAL(Mach_Control.An_b.An_Quantited); 
				Mach_Control.DT_b.DT_NightHoughCa:=Mach_Control.DT_b.DT_NightHoughCa+UINT_TO_REAL(Mach_Control.Ca_b.Ca_Quantited); 
				Mach_Control.DT_b.DT_NightHough_U :=Mach_Control.DT_b.DT_NightHough_U+1;
			 END_IF
		 END_IF		
        IF ((HMI_Hour>=0 AND HMI_Hour<8) OR  (HMI_Hour>=20 AND HMI_Hour<=23)) THEN
			 IF rOverhangNG.Q AND NOT  Mach_Control.U.EmptyRunMode AND Blueflaging THEN
				Mach_Control.DT_b.DTJD_NightHough :=Mach_Control.DT_b.DTJD_NightHough+UINT_TO_REAL(Mach_Control.An_b.An_Quantited(*+Mach_Control.Ca_b.Ca_Quantited*))/(UINT_TO_REAL(Par.stDT_date.An_Quantity)(*+UINT_TO_REAL(Par.stDT_date.Ca_Quantity)*)); 
				Mach_Control.DT_b.DTJD_NightHoughAn:=Mach_Control.DT_b.DTJD_NightHoughAn+UINT_TO_REAL(Mach_Control.An_b.An_Quantited); 
				Mach_Control.DT_b.DTJD_NightHoughCa:=Mach_Control.DT_b.DTJD_NightHoughCa+UINT_TO_REAL(Mach_Control.Ca_b.Ca_Quantited); 
				Mach_Control.DT_b.DTJD_NightHough_U :=Mach_Control.DT_b.DTJD_NightHough_U+1;
			 END_IF
		 END_IF 
//白班对齐度NG数清零	
        IF DayClear1.Q THEN
			Mach_Control.DT_b.DT_DayHough :=0;
			Mach_Control.DT_b.DT_DayHoughAn:=0;
			Mach_Control.DT_b.DT_DayHoughCa:=0;
			Mach_Control.DT_b.DT_DayHough_U :=0;
			Mach_Control.DT_b.DTJD_DayHough :=0;
			Mach_Control.DT_b.DTJD_DayHoughAn:=0;
			Mach_Control.DT_b.DTJD_DayHoughCa:=0;
			Mach_Control.DT_b.DTJD_DayHough_U :=0;
		END_IF
//晚班对齐度NG数清零	
        IF  NightClear1.Q THEN
			Mach_Control.DT_b.DT_NightHough :=0;
			Mach_Control.DT_b.DT_NightHoughAn:=0;
			Mach_Control.DT_b.DT_NightHoughCa:=0;
			Mach_Control.DT_b.DT_NightHough_U :=0;
			Mach_Control.DT_b.DTJD_NightHough :=0;
			Mach_Control.DT_b.DTJD_NightHoughAn:=0;
			Mach_Control.DT_b.DTJD_NightHoughCa:=0;
			Mach_Control.DT_b.DTJD_NightHough_U :=0;
		END_IF		
		
//对齐度NG下料时间		
        Mach_Control.DT_b.DT_OverhangNG:= DP_Step0=6040 AND   Mach_Control.U.DT_iMode=1 AND  TailCurlStep3>=1000 AND TailCurlStep3<=1180  ;
	
//更换隔膜时间	
		IF Mach_Control.DT_b.Error[24] OR Mach_Control.DT_b.Error[61]	OR Bnt_Blueflaging THEN
			Mach_Control.DT_b.DT_GMchange:=TRUE;
 		END_IF		
		
		IF  Mach_Control.DT_b.DT_GMchange  AND NOT Bnt_Blueflaging (*AND   Mach_Control.U.DT_iMode=1*) AND 
             Mach_Control.DT_b.fWindDiameter>Par.stDT_date.fDiameterWarn     AND   Mach_Control.DT_b.bTensionOK    THEN
			Mach_Control.DT_b.DT_GMchange:=FALSE;
		END_IF
END_ACTION

ACTION _01DT_Auto:
Scan_TON	[1](IN:= , PT:=T#200MS , Q=> , ET=> );//取放料时位置判断正极用
Scan_TON	[2](IN:= , PT:=T#200MS , Q=> , ET=> );//取放料时位置判断负极用
DT_Ton[6](IN:= , PT:=T#0.3S , Q=> , ET=> );
tDtUse[2](IN:=, PT:=T#5S , Q=> , ET=> );
//DP_Step0----叠片主流程
/////////////////////////

An_RectifydevGohomeTon(IN:= , PT:=T#1S , Q=> , ET=> );//正极纠偏平台回原点延时
Ca_RectifydevGohomeTon(IN:= , PT:=T#1S , Q=> , ET=> );//负极纠偏平台回原点延时
Ca_TON[1](PT:=T#0.5S);//负极拍照结果超时


IF Mach_Control.DT_b.CDD_OverStart_First THEN
	CCD.Over.Start.iPhotoDo:=3;
	Mach_Control.DT_b.CDD_OverStart:=TRUE;
END_IF

//对齐度结果汇总
D:=D+1;
IF D<1 OR D>(Par.stDT_date.An_Quantity+Par.stDT_date.Ca_Quantity) THEN
	D:=1;
END_IF
IF CellMemory[Mach_Control.DT_b.DT_Memory].Overhang_Result[D]=2 OR CellMemory[Mach_Control.DT_b.DT_Memory].Overhang_Result[D]=3 OR  
    CellMemory[Mach_Control.DT_b.DT_Memory].Overhang_Result[D]=4 OR OversequelNG THEN
	Mach_Control.DT_b.DT_Oerhang_Z:=2;
END_IF


//单步启动
rDT_SinStepd(CLK:=Mach_Control.DT_b.DT_Start , Q=> );
IF rDT_SinStepd.Q THEN
	DP_SinStepe:=FALSE;
END_IF

//叠台真空关闭层数
rDtUse[3](CLK:=(Mach_Control.An_b.An_Quantited+Mach_Control.Ca_b.Ca_Quantited)>=Par.stDT_date.DtCountSet[1]);
rDtUse[4](CLK:=Mach_Control.Ca_b.Ca_Quantited=0);
IF rDtUse[4].Q THEN//叠台真空开
	arrCyCtrl[arrCyNo.ElectValveName.DTVacuum].Cmd.bON:=TRUE;
	arrCyCtrl[arrCyNo.ElectValveName.DTVacuum].Cmd.bOFF:=FALSE;
END_IF
IF rDtUse[3].Q THEN//叠台真空关
	arrCyCtrl[arrCyNo.ElectValveName.DTVacuum].Cmd.bON:=FALSE;
	arrCyCtrl[arrCyNo.ElectValveName.DTVacuum].Cmd.bOFF:=TRUE;
END_IF
	

//正、负已叠极片清零
rClearcountR_TRIG(CLK:=Mach_Control.DT_b.ClearCount , Q=> );
IF Mach_Control.U.DT_iMode=3 THEN
	IF rClearcountR_TRIG.Q THEN
		Mach_Control.An_b.An_Quantited :=0;
		Mach_Control.Ca_b.Ca_Quantited :=0;
		Mach_Control.An_b.An_KDQuantited :=0;
		Mach_Control.Ca_b.Ca_KDQuantited:=0;
		Mach_Control.An_b.An_FirstFoldCnt:=0;
		Mach_Control.Ca_b.Ca_FirstFoldCnt:=0;
		bFirstFoldFinish[1]:=FALSE;//首层隔膜空叠
		bEmptyFoldMark[1]:=FALSE;//进入空叠流程
		Mach_Control.DT_b.OffloadDone:=FALSE;
		Mach_Control.DT_b.OffloadRequest:=FALSE;//叠电芯完成，请求下电芯
		MEMSET(ADR(CellMemory[Mach_Control.DT_b.DT_Memory]),0,SIZEOF(CellMemory[Mach_Control.DT_b.DT_Memory]));
		Mach_Control.DT_b.DT_Oerhang_Z:=0;
		DP_Step0:=0;
////////////////////////////////////////////////////////////////////////////////////////////////////////////				
		Ca_GohomeDone:=FALSE;
		An_GohomeDone:=FALSE; 
		DTIniti_Done :=FALSE;
		//Ca_BeltGohomeDone :=FALSE;	
////////////////////////////////////////////////////////////////////////////////////////////////////////////
	END_IF
END_IF
IF Mach_Control.Ca_b.Ca_Quantited =0 AND Mach_Control.An_b.An_Quantited =0 AND Mach_Control.An_b.An_KDQuantited =0 AND Mach_Control.Ca_b.Ca_KDQuantited =0 THEN
	Mach_Control.DT_b.OffloadDone:=FALSE;
	Mach_Control.DT_b.OffloadRequest:=FALSE;//叠电芯完成，请求下电芯
END_IF

//对齐度检测复位
tMach_Control_TON(IN:=Mach_Control.DT_b.CDD_OverStart , PT:=T#0.05S , Q=> , ET=> );
IF tMach_Control_TON.Q THEN
	Mach_Control.DT_b.CDD_OverStart:=FALSE;
END_IF
//主轴启动超时报警延时
VirMain_TON(IN:= , PT:=T#5S , Q=> , ET=> );

//接带检测或隔膜色标、、空叠隔膜踢废
BulebntR_TRIG(CLK:=(Mach_Control.DT_b.stBnt_Blueflag OR arrCyCtrl[arrCyNo.CylinderName.PoleInflationCy].Status.OFFState)  AND NOT  Mach_Control.DT_b.DT_Blue_TF, Q=> );//OR Mach_Control.se.Yellowmark    OR Mach_Control.btn.PoleInflationbtn
YellowmarkR_TRIG(CLK:=(Mach_Control.se.Yellowmark)  AND NOT  Mach_Control.DT_b.DT_Blue_TF AND NOT  Mach_Control.DT_b.Yellowmark_TF, Q=> );

IF BulebntR_TRIG.Q AND NOT Bnt_Blueflaging THEN//正常接带空叠隔膜层数
	Bnt_Blueflaging:=TRUE;
	//Mach_Control.An_b.An_Blueflaging_TF:=Mach_Control.An_b.An_BlueflagingKDSet;
	Mach_Control.An_b.An_Blueflaging_TF:=Mach_Control.Ca_b.Ca_Blueflaging_TF:=Par.stDT_date.Ca_BlueflagingKDSet;	
ELSIF YellowmarkR_TRIG.Q AND NOT Bnt_Blueflaging THEN//色标感应器空叠隔膜层数
	Bnt_Blueflaging:=TRUE;
	Mach_Control.DT_b.Error_tips[4]:=TRUE;//检测到蓝标，叠台空叠
	//Mach_Control.An_b.An_Blueflaging_TF:=Mach_Control.An_b.An_YellowmarkKDSet;
	Mach_Control.An_b.An_Blueflaging_TF:=Mach_Control.Ca_b.Ca_Blueflaging_TF:=Par.stDT_date.Ca_YellowmarkKDSet;	
END_IF
IF NOT Bnt_Blueflaging THEN
	Mach_Control.DT_b.Error_tips[4]:=FALSE;//检测到蓝标，叠台空叠
END_IF

IF arrCyCtrl[arrCyNo.CylinderName.PoleInflationCy].Status.OFFState THEN
	Mach_Control.DT_b.BlueflagBnt_Warm:=TRUE;//隔膜气胀轴松开提示是否换卷，需要开启接带踢废
ELSIF stSysState.hmiReset OR Bnt_Blueflaging THEN
	Mach_Control.DT_b.BlueflagBnt_Warm:=FALSE;//隔膜气胀轴松开提示是否换卷，需要开启接带踢废
END_IF


//梯度起步
VirMain_TagatTime:=Par.stDT_date.SinglePosTime-0.025;
IF Mach_Control.Ca_b.Ca_Quantited<1 THEN
	arrAxisCtrl[AxiseNo.VirAxisName.VirMain].Cmd.fOverride:=30;
ELSIF  Mach_Control.An_b.An_Quantited<3 OR 
         ((An_OverNGStep>1000 OR Ca_OverNGStep>1000 )(*AND  arrAxis[AxiseNo.VirAxisName.VirMain].Status.NotMoving	*)) OR 
         (Mach_Control.Ca_b.Ca_Quantited= Par.stDT_date.Ca_Quantity  AND Mach_Control.An_b.An_Quantited= Par.stDT_date.An_Quantity)  THEN
	arrAxisCtrl[AxiseNo.VirAxisName.VirMain].Cmd.fOverride:=50;	
ELSIF  Mach_Control.An_b.An_Quantited<4 AND NOT An_OverNGMark AND NOT Ca_OverNGMark  THEN
	arrAxisCtrl[AxiseNo.VirAxisName.VirMain].Cmd.fOverride:=80;
ELSE
	arrAxisCtrl[AxiseNo.VirAxisName.VirMain].Cmd.fOverride:=100;	
END_IF

//Mach_Control.DT_b.DP_Mode:=TRUE;
IF Mach_Control.DT_b.DP_Mode THEN
		IF Mach_Control.Ca_b.Ca_Quantited>= Par.stDT_date.Ca_Quantity-1 AND Mach_Control.An_b.An_Quantited= Par.stDT_date.An_Quantity AND
			Mach_Control.Ca_b.Ca_Quantited < Par.stDT_date.Ca_Quantity AND Par.stDT_date.An_Quantity<>0  AND Par.stDT_date.Ca_Quantity <>0 AND NOT  Mach_Control.U.EmptyRunMode  THEN
			DP_CheseCam:=TRUE;
		//ELSE
			//DP_CheseCam:=FALSE;
		END_IF
END_IF	


//空叠隔膜时关闭负极叠片搬运真空，防止吸极耳
IF DP_CheseCam THEN
	IF Mach_Control.Ca_b.Ca_Quantited>=Par.stDT_date.Ca_Quantity THEN
		arrCyCtrl[arrCyNo.ElectValveName.CaDTCarryingVacuum].Cmd.bON:=TRUE;//负极叠片搬运升降真空破
		arrCyCtrl[arrCyNo.ElectValveName.CaDTCarryingVacuum].Cmd.bOFF:=FALSE;//负极叠片搬运升降真空破
	END_IF
END_IF

//接带或黄标空叠隔膜时,负极搬运破真空，防止吸极耳
IF (Bnt_Blueflaging OR Mach_Control.DT_b.DT_Oerhang_Z=2) AND KD_Mark THEN
	arrCyCtrl[arrCyNo.ElectValveName.CaDTCarryingVacuum].Cmd.bON:=TRUE;//负极叠片搬运升降真空破
	arrCyCtrl[arrCyNo.ElectValveName.CaDTCarryingVacuum].Cmd.bOFF:=FALSE;//负极叠片搬运升降真空破
END_IF

IF Mach_Control.U.DT_iMode=1 THEN//在自动状态下
//叠片自动程序
//CASE DP_Step0 OF
//0://根据已叠正、负极片数来判断当前是需要正极片还是负极片
IF  DP_Step0=0 THEN    	
	IF NOT DP_SinStepe THEN		
		PosErrorMark:=FALSE;
		IF iTensionAutoStep=6666 AND DTPosError[10] THEN//上张力完成
			arrAxisCtrl[AxiseNo.VirAxisName.VirMain].Cmd.bMoveAbs:=FALSE;
			fAnScaling:=1;//20240508 CF
			fCaScaling:=1;//20240508 CF			
			IF NOT Mach_Control.DT_b.FirstEmpFold AND Mach_Control.An_b.An_Quantited=0 AND Mach_Control.Ca_b.Ca_Quantited=0  
				AND Mach_Control.An_b.An_FirstFoldCnt<Mach_Control.An_b.An_FirstFoldSet  AND Mach_Control.An_b.An_FirstFoldSet<>0
				AND Mach_Control.Ca_b.Ca_FirstFoldCnt<Mach_Control.Ca_b.Ca_FirstFoldSet AND Mach_Control.Ca_b.Ca_FirstFoldSet<>0 
				AND NOT bFirstFoldFinish[1] AND NOT bEmptyFoldMark[1]AND An_OverNGStep=0 AND Ca_OverNGStep=0 THEN   //新增，首层隔膜
				Mach_Control.DTRunStatus.bJumpSync:=TRUE;//20240504 CF
				iEmptyFoldStep[1]:=100;//进入首层空叠隔膜流程
				GMlappos[1]:=arrAxisCtrl[AxiseNo.AxisName.SEPTAunwinding].Status.fActPos;
				DP_Step0:=1;
				
			ELSIF NOT Bnt_Blueflaging 
				AND  Mach_Control.An_b.An_Quantited >= Par.stDT_date.An_Quantity  
				AND  Mach_Control.Ca_b.Ca_Quantited >= Par.stDT_date.Ca_Quantity 
				AND Par.stDT_date.An_Quantity<>0  
				AND Par.stDT_date.Ca_Quantity <>0 
				AND iEmptyFoldStep[1]=0 AND An_OverNGStep=0 AND Ca_OverNGStep=0
				(*AND((NOT Mach_Control.DT_b.FirstEmpFold AND bFirstFoldFinish[1])OR(Mach_Control.DT_b.FirstEmpFold))*) THEN//判断当前已叠正、负极片数量是否小于设定的极片数
				//DP_CheseCam:=FALSE;		
				//DP_AnNumber:=0;
				//DP_CaNumber:=0;
				Mach_Control.DTRunStatus.bJumpSync:=TRUE;//20240504 CF
				
				IF NOT  Mach_Control.U.EmptyRunMode THEN
					IF  ( (Mach_Control.An_b.An_KDQuantited >= Par.stDT_date.An_KDQuantity AND  Mach_Control.Ca_b.Ca_KDQuantited  >= Par.stDT_date.Ca_KDQuantity AND Par.stDT_date.An_KDQuantity<>0  AND Par.stDT_date.Ca_KDQuantity<>0 AND Mach_Control.DT_b.DP_Mode ) OR 
						NOT Mach_Control.DT_b.DP_Mode)  THEN
						KD_Mark:=FALSE;//复位空叠隔膜信号
						DP_CheseCam:=FALSE;										
						DP_Step0:=6000;//跳入电芯下料
						GMlappos[2]:=arrAxisCtrl[AxiseNo.AxisName.SEPTAunwinding].Status.fActPos;
						 GMlappos[4]:=GMlappos[2]-GMlappos[1];
						IF ABS(GMlappos[2]-GMlappos[1]) <> 0 THEN
						   GMlappos[3]:=((Mach_Control.An_b.An_Quantited+Mach_Control.Ca_b.Ca_Quantited+3)*par.stDT_date.Width)/ABS(GMlappos[2]-GMlappos[1]);					
						END_IF							
						
					ELSE//电芯空叠尾层隔膜	
						An_Step0:=0;
						An_Step1:=0;
						An_Step2:=0;
						An_Step3:=0;
						An_StandbyStep1:=0;													
						DP_Step0:=1000;//跳入空叠隔膜
					END_IF	
				ELSE//空跑模式	
					Blueflaging:=TRUE;
					Mach_Control.DT_b.Overhang_TF:=TRUE;		
					DP_Step0:=6000;//跳入电芯下料
				END_IF
				
		
			//接带空叠隔膜	
			ELSIF Bnt_Blueflaging AND ((Mach_Control.An_b.An_Quantited=0 AND Mach_Control.Ca_b.Ca_Quantited=0) OR Mach_Control.Ca_b.Ca_Quantited>Mach_Control.An_b.An_Quantited) AND  Par.stDT_date.An_Quantity<>0  
				AND Par.stDT_date.Ca_Quantity <>0 AND Mach_Control.Ca_b.Ca_Quantited>=Par.stDT_date.DT_Overhang_SUM AND Par.stDT_date.DT_Overhang_SUM>0 
                AND iEmptyFoldStep[1]=0 AND An_OverNGStep=0 AND Ca_OverNGStep=0 THEN	
					Mach_Control.DTRunStatus.bJumpSync:=TRUE;//20240504 CF	
					IF Mach_Control.An_b.An_KDQuantited >=Mach_Control.An_b.An_Blueflaging_TF  AND Mach_Control.Ca_b.Ca_KDQuantited >Mach_Control.Ca_b.Ca_Blueflaging_TF  AND Mach_Control.An_b.An_KDQuantited<=Mach_Control.Ca_b.Ca_KDQuantited 
					(*AND((NOT Mach_Control.DT_b.FirstEmpFold AND   bFirstFoldFinish[1]) OR (Mach_Control.DT_b.FirstEmpFold)  )*)  THEN
						Mach_Control.DT_b.Overhang_TF:=TRUE;													
						DT_Ca_Quantited:=0;
						Blueflaging:=TRUE;
						Bnt_Blueflaging:=FALSE;
						KD_Mark:=FALSE;//复位空叠隔膜信号		
						DP_CheseCam:=FALSE;				
						DP_Step0:=6000;//跳入电芯下料
					ELSE//电芯空叠尾层隔膜
						An_Step0:=0;
						An_Step1:=0;
						An_Step2:=0;
						An_Step3:=0;
						An_StandbyStep1:=0;															
						DP_Step0:=1000;//跳入空叠隔膜
					END_IF	
			//对齐度踢废																										
			ELSIF   Mach_Control.An_b.An_Quantited<Mach_Control.Ca_b.Ca_Quantited AND Par.stDT_date.An_Quantity<>0  
				AND Par.stDT_date.Ca_Quantity <>0 AND  Mach_Control.DT_b.DT_CellNG_TF 
				AND (arrAxisCtrl[AxiseNo.AxisName.SEPTATLine].Cmd.arrbRealPoint[1] OR (arrAxisCtrl[AxiseNo.AxisName.SEPTATLine].Cmd.arrbRealPoint[2] AND Mach_Control.An_b.An_KDQuantited >= 1))
				AND	Mach_Control.Ca_b.Ca_Quantited>=Par.stDT_date.DT_Overhang_SUM AND Par.stDT_date.DT_Overhang_SUM>0
				AND Mach_Control.DT_b.DT_Oerhang_Z=2 AND  NOT Mach_Control.U.EmptyRunMode AND NOT Mach_Control.DT_b.DT_Overhang
				AND iEmptyFoldStep[1]=0 AND An_OverNGStep=0 AND Ca_OverNGStep=0
				(*AND((NOT Mach_Control.DT_b.FirstEmpFold AND   bFirstFoldFinish[1]) OR (Mach_Control.DT_b.FirstEmpFold)  )*)  THEN
				Mach_Control.DTRunStatus.bJumpSync:=TRUE;//20240504 CF
				IF  ( (Mach_Control.An_b.An_KDQuantited >= 1 AND  Mach_Control.Ca_b.Ca_KDQuantited  >= 1
					AND Par.stDT_date.An_KDQuantity<>0  AND Par.stDT_date.Ca_KDQuantity<>0 AND Mach_Control.DT_b.DP_Mode ) OR NOT Mach_Control.DT_b.DP_Mode)  THEN
						KD_Mark:=FALSE;//空叠隔膜中	
						DP_CheseCam:=FALSE;				
						OversequelNG:=FALSE;	
						DP_Step0:=6000;//跳入电芯下料
						Mach_Control.DT_b.Overhang_TF:=TRUE;//
						 GMlappos[2]:=arrAxisCtrl[AxiseNo.AxisName.SEPTAunwinding].Status.fActPos;
						 GMlappos[4]:=GMlappos[2]-GMlappos[1];
						IF ABS(GMlappos[2]-GMlappos[1]) <> 0 THEN
						    GMlappos[3]:=((Mach_Control.An_b.An_Quantited+Mach_Control.Ca_b.Ca_Quantited+3)*par.stDT_date.Width)/ABS(GMlappos[2]-GMlappos[1]);	
						END_IF						
						
				ELSE
					An_Step0:=0;
					An_Step1:=0;
					An_Step2:=0;
					An_Step3:=0;
					An_StandbyStep1:=0;													
					DP_Step0:=1000;//跳入空叠隔膜
				END_IF		
				
			ELSE//判断叠负极片还是正极片
				Mach_Control.DTRunStatus.bJumpSync:=FALSE;//20240504 CF
				DT_Ton[6].IN:=FALSE;
				IF Mach_Control.Ca_b.Ca_Quantited = Mach_Control.An_b.An_Quantited AND iEmptyFoldStep[1]=0 AND An_OverNGStep=0 AND Ca_OverNGStep=0 (*AND((NOT Mach_Control.DT_b.FirstEmpFold AND   bFirstFoldFinish[1]) OR Mach_Control.DT_b.FirstEmpFold )*) THEN
					IF Mach_Control.DT_b.SinStepMode THEN//单步调试模式
						DP_SinStepe:=TRUE;
					ELSE
						DP_SinStepe:=FALSE;	
					END_IF		
						Ca_Number:=FALSE;
					IF 	 Mach_Control.Ca_b.Ca_Quantited=0 THEN
						Mach_Control.DT_b.DT_Oerhang_Z:=0;
						MEMSET(ADR(CellMemory[Mach_Control.DT_b.DT_Memory]),0,SIZEOF(CellMemory[Mach_Control.DT_b.DT_Memory]));
					END_IF	
					//DP_CaNumber:=DP_CaNumber+1;	
				
	////////////////////////////////////////////////////////////////////////////////////////////////////////////											
						An_Step0:=0;
						An_Step1:=0;
						An_Step2:=0;
						An_Step3:=0;
						An_StandbyStep1:=0;
						An_OverNGStep:=0;
				    	Ca_OverNGStep:=0;
	////////////////////////////////////////////////////////////////////////////////////////////////////////////											
					
					//DP_AnNumber:=0;								
					DP_Step0:=100;//叠负极片
					DPtime:=12;
				ELSIF Mach_Control.Ca_b.Ca_Quantited > Mach_Control.An_b.An_Quantited AND iEmptyFoldStep[1]=0 AND An_OverNGStep=0 AND Ca_OverNGStep=0 (*AND((NOT Mach_Control.DT_b.FirstEmpFold AND   bFirstFoldFinish[1]) OR (Mach_Control.DT_b.FirstEmpFold)  )*) THEN
					IF Mach_Control.DT_b.SinStepMode THEN
						DP_SinStepe:=TRUE;
					ELSE
						DP_SinStepe:=FALSE;
					END_IF
					An_Number:=FALSE;
					//DP_AnNumber:=DP_AnNumber+1;
					
	////////////////////////////////////////////////////////////////////////////////////////////////////////////													
					Ca_Step0:=0;//负极搬运子程序1
					Ca_Step1:=0;//负极搬运子程序2
					Ca_Step2:=0;//负极搬运子程序3
					Ca_Step3:=0;//负极搬运子程序4		
					Ca_StandbyStep0:=0;
					An_OverNGStep:=0;
					Ca_OverNGStep:=0;
	////////////////////////////////////////////////////////////////////////////////////////////////////////////																	
					//DP_CaNumber:=0;
					DP_Step0:=500;//叠正极片
					DPtime:=22;
				END_IF
			END_IF
		
		ELSIF NOT DTPosError[10] THEN
			Mach_Control.DT_b.Error[60]:=TRUE;//主轴启动前轴有故障
		END_IF
	END_IF
END_IF	
//100://判断负极取料是否完成
IF  DP_Step0=100 THEN 
	IF NOT DP_SinStepe THEN
		IF (Mach_Control.Ca_b.Ca_CarryingFalg AND  Mach_Control.Ca_b.Ca_DPCarryingFalg  
		 AND (CCD.CaRec.Finish.RectifyResult=1 OR  Mach_Control.U.CCD_ChosesHMI OR Mach_Control.U.EmptyRunMode))   THEN//负极取极片OK
			Mach_Control.Ca_b.Ca_DPRequest:=FALSE;//负极极片备料请求
			IF (*Mach_Control.Ca_b.Ca_deviationFPOK AND *) TailCurlSEPTA_SafePos   THEN//
				IF Mach_Control.DT_b.SinStepMode THEN//单步调试模式
					DP_SinStepe:=TRUE;
				ELSE
					DP_SinStepe:=FALSE;	
				END_IF												
				DP_Step0:=101;
				DPtime:=13;
			END_IF
		ELSE
			Mach_Control.DTRunStatus.bJumpSync:=TRUE;//20240509 CF
			IF Ca_StandbyStep0=6666 OR Ca_StandbyStep0=0 THEN
				Ca_StandbyStep0:=1000;//调用负极取片子程序
			END_IF
			IF Mach_Control.DT_b.SinStepMode THEN//单步调试模式
				DP_SinStepe:=TRUE;
			ELSE
				DP_SinStepe:=FALSE;	
			END_IF										
			DP_Step0:=103;
		END_IF
	END_IF
END_IF	
//101://判断主轴是否停止、是否在初始位、是否有轴在耦合中
IF  DP_Step0=101 THEN 
	IF NOT DP_SinStepe THEN
		IF arrAxisCtrl[AxiseNo.VirAxisName.VirMain].Status.NoMoving AND arrAxisCtrl[AxiseNo.VirAxisName.VirMain].Status.fSetPos=0 AND NOT DT_AxiseCoupling THEN
			IF Mach_Control.DT_b.SinStepMode THEN//单步调试模式
				DP_SinStepe:=TRUE;
			ELSE
				DP_SinStepe:=FALSE;	
			END_IF								
			DP_Step0:=104;
			DPtime:=14;
		ELSIF DP_Step1=0 OR DP_Step1=6666 THEN
			DP_Step1:=100;//调用主轴回初始位子程序
			DP_Step0:=102;
		END_IF
	END_IF
END_IF
//102://判断主轴的模长的当前位置是否为0
IF  DP_Step0=102 THEN 
	IF DP_Step1=6666 AND arrAxisCtrl[AxiseNo.VirAxisName.VirMain].Status.NoMoving AND arrAxisCtrl[AxiseNo.VirAxisName.VirMain].Status.fSetPos=0 AND NOT DT_AxiseCoupling  THEN
		IF Mach_Control.DT_b.SinStepMode THEN//单步调试模式
			DP_SinStepe:=TRUE;
		ELSE
			DP_SinStepe:=FALSE;	
		END_IF								
		DP_Step0:=104;
	END_IF
END_IF
//103://等待负极取片完成
IF  DP_Step0=103 THEN 
	IF Ca_StandbyStep0 =6666 THEN//正常取料完成
		DP_Step0:=0;
	ELSIF Ca_StandbyStep0 =0 THEN//取料报警返回
		DP_Step0:=0;
	END_IF
END_IF
	

//104://判断NG气缸是否在安全位
IF  DP_Step0=104 THEN 
	IF arrCyCtrl[arrCyNo.CylinderName.AnScrapbinCy].Status.ONState AND arrCyCtrl[arrCyNo.CylinderName.CaScrapbinUDCy].Status.OFFState AND
		arrCyCtrl[arrCyNo.CylinderName.CaScrapbinCy].Status.ONState AND arrCyCtrl[arrCyNo.CylinderName.PreDiaph].Status.OFFState AND 
		arrCyCtrl[arrCyNo.CylinderName.PoleHotCutterCy].Status.OFFState AND arrCyCtrl[arrCyNo.CylinderName.PoleTapeCy].Status.OFFState AND
		arrCyCtrl[arrCyNo.CylinderName.PoleTapeSplicerRCy].Status.ONState AND arrCyCtrl[arrCyNo.CylinderName.PoleTapeSplicerLCy].Status.ONState AND
        (arrAxisCtrl[AxiseNo.AxisName.LeftYDUpDown].Cmd.arrbRealPoint[1] OR (Ca_OverNGMark AND arrAxisCtrl[AxiseNo.AxisName.LeftYDUpDown].Cmd.arrbRealPoint[15]))
         AND arrAxisCtrl[AxiseNo.AxisName.RightYDUpDown].Cmd.arrbRealPoint[1]   THEN
		DP_Step0:=110;		
	ELSE
		DP_Step0:=105;	
	END_IF
END_IF	
//105:
IF  DP_Step0=105 THEN 
		arrCyCtrl[arrCyNo.CylinderName.AnScrapbinCy].Cmd.bON:=TRUE;
		arrCyCtrl[arrCyNo.CylinderName.PreDiaph].Cmd.bOFF:=TRUE;
		arrCyCtrl[arrCyNo.CylinderName.PoleHotCutterCy].Cmd.bOFF:=TRUE;
		arrCyCtrl[arrCyNo.CylinderName.PoleTapeCy].Cmd.bOFF:=TRUE;
		arrCyCtrl[arrCyNo.CylinderName.PoleTapeSplicerRCy].Cmd.bON:=TRUE;
		arrCyCtrl[arrCyNo.CylinderName.PoleTapeSplicerLCy].Cmd.bON:=TRUE;
		arrCyCtrl[arrCyNo.CylinderName.CaScrapbinCy].Cmd.bON:=TRUE;
		IF   arrCyCtrl[arrCyNo.CylinderName.AnScrapbinCy].Status.ONState AND  arrCyCtrl[arrCyNo.CylinderName.PreDiaph].Status.OFFState AND 
			arrCyCtrl[arrCyNo.CylinderName.PoleHotCutterCy].Status.OFFState AND arrCyCtrl[arrCyNo.CylinderName.PoleTapeCy].Status.OFFState AND
			arrCyCtrl[arrCyNo.CylinderName.PoleTapeSplicerRCy].Status.ONState AND arrCyCtrl[arrCyNo.CylinderName.PoleTapeSplicerLCy].Status.ONState
		AND arrCyCtrl[arrCyNo.CylinderName.CaScrapbinCy].Cmd.bON THEN
			DP_Step0:=106;									
		END_IF
END_IF
//106:
IF  DP_Step0=106 THEN 
	arrCyCtrl[arrCyNo.CylinderName.CaScrapbinUDCy].Cmd.bOFF:=TRUE;
	IF  arrCyCtrl[arrCyNo.CylinderName.CaScrapbinUDCy].Status.OFFState AND 
        ( arrAxisCtrl[AxiseNo.AxisName.LeftYDUpDown].Cmd.arrbRealPoint[1]OR (Ca_OverNGMark AND arrAxisCtrl[AxiseNo.AxisName.LeftYDUpDown].Cmd.arrbRealPoint[15])) 
       AND arrAxisCtrl[AxiseNo.AxisName.RightYDUpDown].Cmd.arrbRealPoint[1]  THEN
		DP_Step0:=110;	
	END_IF	
END_IF						
//110:
IF  DP_Step0=110 THEN 
    An_OverhangNG:=FALSE;
	IF NOT DP_SinStepe THEN
		Scan_TON[2].IN:=TRUE;		
		IF CA_CarryingPos1  THEN//负极搬运、叠片各轴在初始位
			Scan_TON[1].IN:=TRUE;	
			IF AN_CarryingPos2  THEN//正极在叠片位
				fAnScaling:=0.8;//20240508 CF	
				IF arrAxisCtrl[AxiseNo.AxisName.SEPTATLine].Cmd.arrbRealPoint[2]   THEN
					//IF Mach_Control.An_b.An_deviationDPOK  THEN//正极纠偏平台,拍照完成
						IF  NOT Mach_Control.An_b.An_DPCarryingFalg AND  Mach_Control.An_b.An_deviationFalg AND NOT DP_CheseCam 
						AND ((NOT Mach_Control.DT_b.FirstEmpFold AND Mach_Control.An_b.An_FirstFoldCnt=Mach_Control.An_b.An_FirstFoldSet  ) OR Mach_Control.DT_b.FirstEmpFold  )
						AND Mach_Control.An_b.An_Quantited< Par.stDT_date.An_Quantity  THEN  //叠片搬运需要取片  AND Mach_Control.An_b.An_deviationDPOK
							iAnCamInSel2:=1;
						ELSE
							iAnCamInSel2:=2;
						END_IF    
  
						Ca_CanIn4:=TRUE;
					
						IF Mach_Control.DT_b.SinStepMode THEN//单步调试模式
							DP_SinStepe:=TRUE;
						ELSE
							DP_SinStepe:=FALSE;	
						END_IF	
						DP_Step0:=160;//
						DPtime:=32;	
					//END_IF
				ELSE
					Mach_Control.DT_b.Error[5]:=TRUE;//叠负极片凸轮耦合时，隔膜平移轴即不在负极叠片位，也不在正极叠片位报警
					DP_Step0:=9991;	
				END_IF;
			ELSIF AN_CarryingPos1  THEN//在取片位	
				Mach_Control.DTRunStatus.bJumpSync:=TRUE;//20240504 CF																			
				IF arrAxisCtrl[AxiseNo.AxisName.SEPTATLine].Cmd.arrbRealPoint[1]  THEN
					IF Mach_Control.DT_b.SinStepMode THEN//单步调试模式
						DP_SinStepe:=TRUE;
					ELSE
						DP_SinStepe:=FALSE;	
					END_IF											
					DP_Step0:=130;//
				ELSIF arrAxisCtrl[AxiseNo.AxisName.SEPTATLine].Cmd.arrbRealPoint[2] THEN
					IF Mach_Control.DT_b.SinStepMode THEN//单步调试模式
						DP_SinStepe:=TRUE;
					ELSE
						DP_SinStepe:=FALSE;	
					END_IF											
					DP_Step0:=140;//
				ELSE
					Mach_Control.DT_b.Error[5]:=TRUE;//叠负极片凸轮耦合时，隔膜平移轴即不在负极叠片位，也不在正极叠片位报警
					DP_Step0:=9992;	
				END_IF;							
			ELSIF Scan_TON[1].Q THEN
				Scan_TON[1].IN:=FALSE;	
				DP_Step0:=9993;
				DTPosError[3]:=TRUE;
			END_IF
	
